LIN {X 0,Y 303.786,Z 846.921,A -85,B 0,C 180,E1 -15924.689,E2 -15924.689} C_VEL
LIN {X 0,Y 303.796,Z 848.766,A -85,B 0,C 180,E1 -15926.019,E2 -15926.019} C_VEL
LIN {X 0,Y 303.768,Z 850.119,A -85,B 0,C 180,E1 -15927.346,E2 -15927.346} C_VEL
LIN {X 0,Y 303.87,Z 851.06,A -85,B 0,C 180,E1 -15928.673,E2 -15928.673} C_VEL
LIN {X 0,Y 303.954,Z 851.584,A -85,B 0,C 180,E1 -15929.999,E2 -15929.999} C_VEL
LIN {X 0,Y 303.824,Z 851.641,A -85,B 0,C 180,E1 -15931.324,E2 -15931.324} C_VEL
LIN {X 0,Y 303.734,Z 851.272,A -85,B 0,C 180,E1 -15932.651,E2 -15932.651} C_VEL
LIN {X 0,Y 303.715,Z 850.5,A -85,B 0,C 180,E1 -15933.979,E2 -15933.979} C_VEL
LIN {X 0,Y 303.689,Z 848.909,A -85,B 0,C 180,E1 -15935.665,E2 -15935.665} C_VEL
LIN {X 0,Y 303.939,Z 845.59,A -85,B 0,C 180,E1 -15937.973,E2 -15937.973} C_VEL
LIN {X 0,Y 304.361,Z 841.592,A -85,B 0,C 180,E1 -15939.971,E2 -15939.971} C_VEL
LIN {X 0,Y 305.048,Z 836.47,A -85,B 0,C 180,E1 -15941.966,E2 -15941.966} C_VEL
LIN {X 0,Y 306.228,Z 830.072,A -85,B 0,C 180,E1 -15943.943,E2 -15943.943} C_VEL
LIN {X 0,Y 307.615,Z 822.158,A -85,B 0,C 180,E1 -15945.91,E2 -15945.91} C_VEL
LIN {X 0,Y 309.269,Z 812.287,A -85,B 0,C 180,E1 -15947.864,E2 -15947.864} C_VEL
LIN {X 0,Y 311.114,Z 802.166,A -85,B 0,C 180,E1 -15949.461,E2 -15949.461} C_VEL
LIN {X 0,Y 312.828,Z 792.253,A -85,B 0,C 180,E1 -15950.721,E2 -15950.721} C_VEL
LIN {X 0,Y 314.602,Z 779.923,A -85,B 0,C 180,E1 -15951.972,E2 -15951.972} C_VEL
LIN {X 0,Y 316.384,Z 766.923,A -85,B 0,C 180,E1 -15952.961,E2 -15952.961} C_VEL
LIN {X 0,Y 317.699,Z 753.709,A -85,B 0,C 180,E1 -15953.679,E2 -15953.679} C_VEL
LIN {X 0,Y 318.529,Z 740.017,A -85,B 0,C 180,E1 -15954.176,E2 -15954.176} C_VEL
LIN {X 0,Y 320.65,Z 684.229,A -85,B 0,C 180,E1 -15955.689,E2 -15955.689} C_VEL
LIN {X 0,Y 318.484,Z 666.248,A -85,B 0,C 180,E1 -15956.514,E2 -15956.514} C_VEL
LIN {X 0,Y 315.684,Z 649.939,A -85,B 0,C 180,E1 -15957.399,E2 -15957.399} C_VEL
LIN {X 0,Y 312.951,Z 638.201,A -85,B 0,C 180,E1 -15958.147,E2 -15958.147} C_VEL
LIN {X 0,Y 312.146,Z 635.73,A -85,B 0,C 180,E1 -15958.373,E2 -15958.373} C_VEL
LIN {X 0,Y 310.349,Z 626.488,A -85,B 0,C 180,E1 -15961.387,E2 -15961.387} C_VEL
LIN {X 0,Y 308.701,Z 619.358,A -85,B 0,C 180,E1 -15963.9,E2 -15963.9} C_VEL
LIN {X 0,Y 306.797,Z 612.092,A -85,B 0,C 180,E1 -15966.7,E2 -15966.7} C_VEL
LIN {X 0,Y 305.491,Z 607.435,A -85,B 0,C 180,E1 -15968.684,E2 -15968.684} C_VEL
LIN {X 0,Y 305.495,Z 607.433,A -85,B 0,C 180,E1 -15972.594,E2 -15972.594} C_VEL
LIN {X 0,Y 305.497,Z 607.431,A -85,B 0,C 180,E1 -15976.357,E2 -15976.357} C_VEL
LIN {X 0,Y 305.494,Z 607.433,A -85,B 0,C 180,E1 -15979.898,E2 -15979.898} C_VEL
LIN {X 0,Y 305.497,Z 607.426,A -85,B 0,C 180,E1 -15983.625,E2 -15983.625} C_VEL
LIN {X 0,Y 305.46,Z 607.431,A -85,B 0,C 180,E1 -15986.482,E2 -15986.482} C_VEL
LIN {X 0,Y 305.46,Z 607.432,A -85,B 0,C 180,E1 -15989.59,E2 -15989.59} C_VEL
LIN {X 0,Y 305.515,Z 607.427,A -85,B 0,C 180,E1 -15992.608,E2 -15992.608} C_VEL
LIN {X 0,Y 305.501,Z 607.428,A -85,B 0,C 180,E1 -15995.538,E2 -15995.538} C_VEL
LIN {X 0,Y 305.512,Z 607.423,A -85,B 0,C 180,E1 -15999.814,E2 -15999.814} C_VEL
LIN {X 0,Y 305.566,Z 607.418,A -85,B 0,C 180,E1 -16002.602,E2 -16002.602} C_VEL
LIN {X 0,Y 305.641,Z 607.408,A -85,B 0,C 180,E1 -16005.348,E2 -16005.348} C_VEL
LIN {X 0,Y 305.632,Z 607.414,A -85,B 0,C 180,E1 -16009.399,E2 -16009.399} C_VEL
LIN {X 0,Y 305.805,Z 607.392,A -85,B 0,C 180,E1 -16012.074,E2 -16012.074} C_VEL
LIN {X 0,Y 305.682,Z 607.406,A -85,B 0,C 180,E1 -16014.723,E2 -16014.723} C_VEL
LIN {X 0,Y 305.951,Z 607.373,A -85,B 0,C 180,E1 -16018.684,E2 -16018.684} C_VEL
LIN {X 0,Y 305.953,Z 607.376,A -85,B 0,C 180,E1 -16021.316,E2 -16021.316} C_VEL
LIN {X 0,Y 305.658,Z 607.553,A -85,B 0,C 180,E1 -16024.533,E2 -16024.533} C_VEL
LIN {X 0,Y 306.632,Z 610.635,A -85,B 0,C 180,E1 -16025.982,E2 -16025.982} C_VEL
LIN {X 0,Y 313.096,Z 622.289,A -85,B 0,C 180,E1 -16027.316,E2 -16027.316} C_VEL
LIN {X 0,Y 320.199,Z 637.232,A -85,B 0,C 180,E1 -16028.725,E2 -16028.725} C_VEL
LIN {X 0,Y 322.11,Z 641.956,A -85,B 0,C 180,E1 -16029.111,E2 -16029.111} C_VEL
LIN {X 0,Y 319.07,Z 715.822,A -85,B 0,C 180,E1 -16031.152,E2 -16031.152} C_VEL
LIN {X 0,Y 318.2,Z 728.923,A -85,B 0,C 180,E1 -16031.757,E2 -16031.757} C_VEL
LIN {X 0,Y 317.117,Z 741.244,A -85,B 0,C 180,E1 -16032.577,E2 -16032.577} C_VEL
LIN {X 0,Y 315.862,Z 751.913,A -85,B 0,C 180,E1 -16033.511,E2 -16033.511} C_VEL
LIN {X 0,Y 314.2,Z 763.939,A -85,B 0,C 180,E1 -16034.87,E2 -16034.87} C_VEL
LIN {X 0,Y 312.488,Z 774.225,A -85,B 0,C 180,E1 -16036.328,E2 -16036.328} C_VEL
LIN {X 0,Y 310.781,Z 783.569,A -85,B 0,C 180,E1 -16037.98,E2 -16037.98} C_VEL
LIN {X 0,Y 309.046,Z 792.453,A -85,B 0,C 180,E1 -16039.945,E2 -16039.945} C_VEL
LIN {X 0,Y 307.616,Z 799.149,A -85,B 0,C 180,E1 -16041.793,E2 -16041.793} C_VEL
LIN {X 0,Y 306.432,Z 805.122,A -85,B 0,C 180,E1 -16043.896,E2 -16043.896} C_VEL
LIN {X 0,Y 305.394,Z 810.016,A -85,B 0,C 180,E1 -16046.172,E2 -16046.172} C_VEL
LIN {X 0,Y 304.957,Z 812.136,A -85,B 0,C 180,E1 -16047.446,E2 -16047.446} C_VEL
LIN {X 0,Y 304.502,Z 814.135,A -85,B 0,C 180,E1 -16048.992,E2 -16048.992} C_VEL
LIN {X 0,Y 304,Z 815.985,A -85,B 0,C 180,E1 -16051.201,E2 -16051.201} C_VEL
LIN {X 0,Y 303.73,Z 816.702,A -85,B 0,C 180,E1 -16053.734,E2 -16053.734} C_VEL
LIN {X 0,Y 303.63,Z 816.128,A -85,B 0,C 180,E1 -16055.894,E2 -16055.894} C_VEL
LIN {X 0,Y 303.743,Z 814.383,A -85,B 0,C 180,E1 -16058.125,E2 -16058.125} C_VEL
LIN {X 0,Y 304.075,Z 811.449,A -85,B 0,C 180,E1 -16060.327,E2 -16060.327} C_VEL
LIN {X 0,Y 304.45,Z 807.575,A -85,B 0,C 180,E1 -16062.382,E2 -16062.382} C_VEL
LIN {X 0,Y 305.045,Z 802.499,A -85,B 0,C 180,E1 -16064.423,E2 -16064.423} C_VEL
LIN {X 0,Y 305.768,Z 796.24,A -85,B 0,C 180,E1 -16066.408,E2 -16066.408} C_VEL
LIN {X 0,Y 306.705,Z 788.58,A -85,B 0,C 180,E1 -16068.357,E2 -16068.357} C_VEL
LIN {X 0,Y 307.67,Z 780.998,A -85,B 0,C 180,E1 -16069.927,E2 -16069.927} C_VEL
LIN {X 0,Y 308.786,Z 771.91,A -85,B 0,C 180,E1 -16071.479,E2 -16071.479} C_VEL
LIN {X 0,Y 310.089,Z 760.631,A -85,B 0,C 180,E1 -16073.027,E2 -16073.027} C_VEL
LIN {X 0,Y 311.104,Z 749.624,A -85,B 0,C 180,E1 -16074.238,E2 -16074.238} C_VEL
LIN {X 0,Y 312.157,Z 737.533,A -85,B 0,C 180,E1 -16075.263,E2 -16075.263} C_VEL
LIN {X 0,Y 312.912,Z 724.139,A -85,B 0,C 180,E1 -16076.108,E2 -16076.108} C_VEL
LIN {X 0,Y 313.468,Z 711.355,A -85,B 0,C 180,E1 -16076.648,E2 -16076.648} C_VEL
LIN {X 0,Y 315.639,Z 635.414,A -85,B 0,C 180,E1 -16078.638,E2 -16078.638} C_VEL
LIN {X 0,Y 308.701,Z 615.889,A -85,B 0,C 180,E1 -16079.648,E2 -16079.648} C_VEL
LIN {X 0,Y 305.52,Z 607.516,A -85,B 0,C 180,E1 -16080.111,E2 -16080.111} C_VEL
LIN {X 0,Y 305.568,Z 607.425,A -85,B 0,C 180,E1 -16084.089,E2 -16084.089} C_VEL
LIN {X 0,Y 305.527,Z 607.428,A -85,B 0,C 180,E1 -16088.407,E2 -16088.407} C_VEL
LIN {X 0,Y 305.59,Z 607.416,A -85,B 0,C 180,E1 -16091.219,E2 -16091.219} C_VEL
LIN {X 0,Y 305.648,Z 607.409,A -85,B 0,C 180,E1 -16095.351,E2 -16095.351} C_VEL
LIN {X 0,Y 305.64,Z 607.41,A -85,B 0,C 180,E1 -16099.401,E2 -16099.401} C_VEL
LIN {X 0,Y 305.813,Z 607.391,A -85,B 0,C 180,E1 -16102.076,E2 -16102.076} C_VEL
LIN {X 0,Y 305.69,Z 607.407,A -85,B 0,C 180,E1 -16104.725,E2 -16104.725} C_VEL
LIN {X 0,Y 305.957,Z 607.375,A -85,B 0,C 180,E1 -16108.685,E2 -16108.685} C_VEL
LIN {X 0,Y 305.961,Z 607.37,A -85,B 0,C 180,E1 -16111.318,E2 -16111.318} C_VEL
LIN {X 0,Y 305.692,Z 607.404,A -85,B 0,C 180,E1 -16115.278,E2 -16115.278} C_VEL
LIN {X 0,Y 305.815,Z 607.388,A -85,B 0,C 180,E1 -16117.927,E2 -16117.927} C_VEL
LIN {X 0,Y 305.606,Z 607.414,A -85,B 0,C 180,E1 -16121.946,E2 -16121.946} C_VEL
LIN {X 0,Y 305.64,Z 607.413,A -85,B 0,C 180,E1 -16125.036,E2 -16125.036} C_VEL
LIN {X 0,Y 305.579,Z 607.416,A -85,B 0,C 180,E1 -16129.446,E2 -16129.446} C_VEL
LIN {X 0,Y 305.494,Z 607.433,A -85,B 0,C 180,E1 -16133.043,E2 -16133.043} C_VEL
LIN {X 0,Y 305.529,Z 607.424,A -85,B 0,C 180,E1 -16136.22,E2 -16136.22} C_VEL
LIN {X 0,Y 305.492,Z 607.434,A -85,B 0,C 180,E1 -16139.049,E2 -16139.049} C_VEL
LIN {X 0,Y 305.445,Z 607.432,A -85,B 0,C 180,E1 -16141.953,E2 -16141.953} C_VEL
LIN {X 0,Y 305.466,Z 607.433,A -85,B 0,C 180,E1 -16145.114,E2 -16145.114} C_VEL
LIN {X 0,Y 305.444,Z 607.434,A -85,B 0,C 180,E1 -16148.528,E2 -16148.528} C_VEL
LIN {X 0,Y 305.463,Z 607.432,A -85,B 0,C 180,E1 -16152.587,E2 -16152.587} C_VEL
LIN {X 0,Y 305.447,Z 607.433,A -85,B 0,C 180,E1 -16156.349,E2 -16156.349} C_VEL
LIN {X 0,Y 305.462,Z 607.431,A -85,B 0,C 180,E1 -16159.893,E2 -16159.893} C_VEL
LIN {X 0,Y 305.454,Z 607.429,A -85,B 0,C 180,E1 -16162.054,E2 -16162.054} C_VEL
LIN {X 0,Y 304.762,Z 607.519,A -85,B 0,C 180,E1 -16163.155,E2 -16163.155} C_VEL
LIN {X 0,Y 301.888,Z 607.875,A -85,B 0,C 180,E1 -16164.947,E2 -16164.947} C_VEL
LIN {X 0,Y 299.48,Z 608.175,A -85,B 0,C 180,E1 -16166.4,E2 -16166.4} C_VEL
LIN {X 0,Y 298.47,Z 608.306,A -85,B 0,C 180,E1 -16167.526,E2 -16167.526} C_VEL
LIN {X 0,Y 298.399,Z 608.313,A -85,B 0,C 180,E1 -16167.907,E2 -16167.907} C_VEL
LIN {X 0,Y 298.469,Z 608.307,A -85,B 0,C 180,E1 -16171.905,E2 -16171.905} C_VEL
LIN {X 0,Y 298.489,Z 608.301,A -85,B 0,C 180,E1 -16174.925,E2 -16174.925} C_VEL
LIN {X 0,Y 298.443,Z 608.306,A -85,B 0,C 180,E1 -16179.315,E2 -16179.315} C_VEL
LIN {X 0,Y 298.54,Z 608.292,A -85,B 0,C 180,E1 -16182.18,E2 -16182.18} C_VEL
LIN {X 0,Y 298.599,Z 608.282,A -85,B 0,C 180,E1 -16184.995,E2 -16184.995} C_VEL
LIN {X 0,Y 298.598,Z 608.286,A -85,B 0,C 180,E1 -16189.147,E2 -16189.147} C_VEL
LIN {X 0,Y 298.747,Z 608.272,A -85,B 0,C 180,E1 -16191.886,E2 -16191.886} C_VEL
LIN {X 0,Y 298.662,Z 608.28,A -85,B 0,C 180,E1 -16194.599,E2 -16194.599} C_VEL
LIN {X 0,Y 298.928,Z 608.245,A -85,B 0,C 180,E1 -16198.653,E2 -16198.653} C_VEL
LIN {X 0,Y 298.928,Z 608.242,A -85,B 0,C 180,E1 -16201.347,E2 -16201.347} C_VEL
LIN {X 0,Y 298.794,Z 608.264,A -85,B 0,C 180,E1 -16206.754,E2 -16206.754} C_VEL
LIN {X 0,Y 298.642,Z 608.282,A -85,B 0,C 180,E1 -16209.482,E2 -16209.482} C_VEL
LIN {X 0,Y 298.552,Z 608.292,A -85,B 0,C 180,E1 -16213.616,E2 -16213.616} C_VEL
LIN {X 0,Y 298.49,Z 608.303,A -85,B 0,C 180,E1 -16216.412,E2 -16216.412} C_VEL
LIN {X 0,Y 298.466,Z 608.304,A -85,B 0,C 180,E1 -16219.627,E2 -16219.627} C_VEL
LIN {X 0,Y 298.435,Z 608.307,A -85,B 0,C 180,E1 -16223.6,E2 -16223.6} C_VEL
LIN {X 0,Y 298.498,Z 608.303,A -85,B 0,C 180,E1 -16226.574,E2 -16226.574} C_VEL
LIN {X 0,Y 298.427,Z 608.309,A -85,B 0,C 180,E1 -16229.641,E2 -16229.641} C_VEL
LIN {X 0,Y 298.401,Z 608.316,A -85,B 0,C 180,E1 -16232.8,E2 -16232.8} C_VEL
LIN {X 0,Y 298.45,Z 608.311,A -85,B 0,C 180,E1 -16236.806,E2 -16236.806} C_VEL
LIN {X 0,Y 298.394,Z 608.317,A -85,B 0,C 180,E1 -16241.087,E2 -16241.087} C_VEL
LIN {X 0,Y 298.394,Z 608.318,A -85,B 0,C 180,E1 -16245.041,E2 -16245.041} C_VEL
LIN {X 0,Y 298.393,Z 608.317,A -85,B 0,C 180,E1 -16248.911,E2 -16248.911} C_VEL
LIN {X 0,Y 298.45,Z 608.311,A -85,B 0,C 180,E1 -16253.192,E2 -16253.192} C_VEL
LIN {X 0,Y 298.448,Z 608.42,A -85,B 0,C 180,E1 -16255.751,E2 -16255.751} C_VEL
LIN {X 0,Y 301.082,Z 620.831,A -85,B 0,C 180,E1 -16259.479,E2 -16259.479} C_VEL
LIN {X 0,Y 303.19,Z 630.91,A -85,B 0,C 180,E1 -16262.379,E2 -16262.379} C_VEL
LIN {X 0,Y 303.241,Z 633.696,A -85,B 0,C 180,E1 -16263.131,E2 -16263.131} C_VEL
LIN {X 0,Y 302.442,Z 639.311,A -85,B 0,C 180,E1 -16264.586,E2 -16264.586} C_VEL
LIN {X 0,Y 308.114,Z 684.772,A -85,B 0,C 180,E1 -16266.296,E2 -16266.296} C_VEL
LIN {X 0,Y 306.225,Z 749.237,A -85,B 0,C 180,E1 -16268.057,E2 -16268.057} C_VEL
LIN {X 0,Y 305.404,Z 762.213,A -85,B 0,C 180,E1 -16268.66,E2 -16268.66} C_VEL
LIN {X 0,Y 304.335,Z 774.343,A -85,B 0,C 180,E1 -16269.467,E2 -16269.467} C_VEL
LIN {X 0,Y 303.101,Z 786.172,A -85,B 0,C 180,E1 -16270.529,E2 -16270.529} C_VEL
LIN {X 0,Y 301.763,Z 797.631,A -85,B 0,C 180,E1 -16271.849,E2 -16271.849} C_VEL
LIN {X 0,Y 300.511,Z 808.02,A -85,B 0,C 180,E1 -16273.351,E2 -16273.351} C_VEL
LIN {X 0,Y 299.442,Z 817.358,A -85,B 0,C 180,E1 -16275.037,E2 -16275.037} C_VEL
LIN {X 0,Y 298.326,Z 826.437,A -85,B 0,C 180,E1 -16277.066,E2 -16277.066} C_VEL
LIN {X 0,Y 297.485,Z 833.693,A -85,B 0,C 180,E1 -16279.104,E2 -16279.104} C_VEL
LIN {X 0,Y 297.018,Z 839.454,A -85,B 0,C 180,E1 -16281.151,E2 -16281.151} C_VEL
LIN {X 0,Y 296.789,Z 843.951,A -85,B 0,C 180,E1 -16283.199,E2 -16283.199} C_VEL
LIN {X 0,Y 296.701,Z 846.302,A -85,B 0,C 180,E1 -16284.562,E2 -16284.562} C_VEL
LIN {X 0,Y 296.727,Z 848.202,A -85,B 0,C 180,E1 -16285.924,E2 -16285.924} C_VEL
LIN {X 0,Y 296.688,Z 849.596,A -85,B 0,C 180,E1 -16287.283,E2 -16287.283} C_VEL
LIN {X 0,Y 296.778,Z 850.566,A -85,B 0,C 180,E1 -16288.642,E2 -16288.642} C_VEL
LIN {X 0,Y 296.867,Z 851.119,A -85,B 0,C 180,E1 -16289.999,E2 -16289.999} C_VEL
LIN {X 0,Y 296.73,Z 851.23,A -85,B 0,C 180,E1 -16291.356,E2 -16291.356} C_VEL
LIN {X 0,Y 296.653,Z 850.888,A -85,B 0,C 180,E1 -16292.714,E2 -16292.714} C_VEL
LIN {X 0,Y 296.626,Z 850.14,A -85,B 0,C 180,E1 -16294.074,E2 -16294.074} C_VEL
LIN {X 0,Y 296.606,Z 848.802,A -85,B 0,C 180,E1 -16295.625,E2 -16295.625} C_VEL
LIN {X 0,Y 296.873,Z 845.348,A -85,B 0,C 180,E1 -16298.164,E2 -16298.164} C_VEL
LIN {X 0,Y 297.348,Z 841.428,A -85,B 0,C 180,E1 -16300.209,E2 -16300.209} C_VEL
LIN {X 0,Y 298.067,Z 836.374,A -85,B 0,C 180,E1 -16302.25,E2 -16302.25} C_VEL
LIN {X 0,Y 299.332,Z 830.045,A -85,B 0,C 180,E1 -16304.271,E2 -16304.271} C_VEL
LIN {X 0,Y 300.792,Z 822.225,A -85,B 0,C 180,E1 -16306.281,E2 -16306.281} C_VEL
LIN {X 0,Y 302.536,Z 812.502,A -85,B 0,C 180,E1 -16308.275,E2 -16308.275} C_VEL
LIN {X 0,Y 304.45,Z 802.56,A -85,B 0,C 180,E1 -16309.905,E2 -16309.905} C_VEL
LIN {X 0,Y 306.493,Z 791.545,A -85,B 0,C 180,E1 -16311.346,E2 -16311.346} C_VEL
LIN {X 0,Y 308.093,Z 780.913,A -85,B 0,C 180,E1 -16312.461,E2 -16312.461} C_VEL
LIN {X 0,Y 310.062,Z 767.228,A -85,B 0,C 180,E1 -16313.545,E2 -16313.545} C_VEL
LIN {X 0,Y 311.36,Z 755.244,A -85,B 0,C 180,E1 -16314.236,E2 -16314.236} C_VEL
LIN {X 0,Y 312.309,Z 741.359,A -85,B 0,C 180,E1 -16314.778,E2 -16314.778} C_VEL
LIN {X 0,Y 314.649,Z 685.473,A -85,B 0,C 180,E1 -16316.333,E2 -16316.333} C_VEL
LIN {X 0,Y 312.673,Z 668.247,A -85,B 0,C 180,E1 -16317.155,E2 -16317.155} C_VEL
LIN {X 0,Y 309.901,Z 651.84,A -85,B 0,C 180,E1 -16318.07,E2 -16318.07} C_VEL
LIN {X 0,Y 307.431,Z 641.003,A -85,B 0,C 180,E1 -16318.792,E2 -16318.792} C_VEL
LIN {X 0,Y 304.991,Z 635.218,A -85,B 0,C 180,E1 -16319.361,E2 -16319.361} C_VEL
LIN {X 0,Y 303.047,Z 625.874,A -85,B 0,C 180,E1 -16322.577,E2 -16322.577} C_VEL
LIN {X 0,Y 301.051,Z 617.638,A -85,B 0,C 180,E1 -16325.704,E2 -16325.704} C_VEL
LIN {X 0,Y 298.78,Z 609.723,A -85,B 0,C 180,E1 -16329.082,E2 -16329.082} C_VEL
LIN {X 0,Y 298.43,Z 608.316,A -85,B 0,C 180,E1 -16329.809,E2 -16329.809} C_VEL
LIN {X 0,Y 298.454,Z 608.311,A -85,B 0,C 180,E1 -16333.114,E2 -16333.114} C_VEL
LIN {X 0,Y 298.462,Z 608.307,A -85,B 0,C 180,E1 -16336.931,E2 -16336.931} C_VEL
LIN {X 0,Y 298.434,Z 608.307,A -85,B 0,C 180,E1 -16340.996,E2 -16340.996} C_VEL
LIN {X 0,Y 298.428,Z 608.307,A -85,B 0,C 180,E1 -16343.931,E2 -16343.931} C_VEL
LIN {X 0,Y 298.393,Z 608.312,A -85,B 0,C 180,E1 -16347.981,E2 -16347.981} C_VEL
LIN {X 0,Y 298.457,Z 608.301,A -85,B 0,C 180,E1 -16351.903,E2 -16351.903} C_VEL
LIN {X 0,Y 298.478,Z 608.302,A -85,B 0,C 180,E1 -16354.923,E2 -16354.923} C_VEL
LIN {X 0,Y 298.451,Z 608.303,A -85,B 0,C 180,E1 -16359.315,E2 -16359.315} C_VEL
LIN {X 0,Y 298.53,Z 608.295,A -85,B 0,C 180,E1 -16362.179,E2 -16362.179} C_VEL
LIN {X 0,Y 298.585,Z 608.287,A -85,B 0,C 180,E1 -16364.994,E2 -16364.994} C_VEL
LIN {X 0,Y 298.587,Z 608.292,A -85,B 0,C 180,E1 -16369.146,E2 -16369.146} C_VEL
LIN {X 0,Y 298.75,Z 608.272,A -85,B 0,C 180,E1 -16371.886,E2 -16371.886} C_VEL
LIN {X 0,Y 298.653,Z 608.281,A -85,B 0,C 180,E1 -16374.599,E2 -16374.599} C_VEL
LIN {X 0,Y 298.917,Z 608.249,A -85,B 0,C 180,E1 -16378.653,E2 -16378.653} C_VEL
LIN {X 0,Y 298.92,Z 608.252,A -85,B 0,C 180,E1 -16381.347,E2 -16381.347} C_VEL
LIN {X 0,Y 298.71,Z 608.484,A -85,B 0,C 180,E1 -16383.541,E2 -16383.541} C_VEL
LIN {X 0,Y 299.47,Z 611.352,A -85,B 0,C 180,E1 -16384.901,E2 -16384.901} C_VEL
LIN {X 0,Y 301.738,Z 615.054,A -85,B 0,C 180,E1 -16385.408,E2 -16385.408} C_VEL
LIN {X 0,Y 307.159,Z 624.505,A -85,B 0,C 180,E1 -16386.569,E2 -16386.569} C_VEL
LIN {X 0,Y 314.123,Z 639.09,A -85,B 0,C 180,E1 -16388.029,E2 -16388.029} C_VEL
LIN {X 0,Y 316.129,Z 643.93,A -85,B 0,C 180,E1 -16388.446,E2 -16388.446} C_VEL
LIN {X 0,Y 312.959,Z 716.358,A -85,B 0,C 180,E1 -16390.513,E2 -16390.513} C_VEL
LIN {X 0,Y 312.01,Z 729.333,A -85,B 0,C 180,E1 -16391.12,E2 -16391.12} C_VEL
LIN {X 0,Y 310.85,Z 742.08,A -85,B 0,C 180,E1 -16391.989,E2 -16391.989} C_VEL
LIN {X 0,Y 309.566,Z 752.553,A -85,B 0,C 180,E1 -16392.929,E2 -16392.929} C_VEL
LIN {X 0,Y 307.93,Z 763.714,A -85,B 0,C 180,E1 -16394.202,E2 -16394.202} C_VEL
LIN {X 0,Y 306.153,Z 774.096,A -85,B 0,C 180,E1 -16395.684,E2 -16395.684} C_VEL
LIN {X 0,Y 304.529,Z 782.271,A -85,B 0,C 180,E1 -16397.112,E2 -16397.112} C_VEL
LIN {X 0,Y 302.774,Z 790.87,A -85,B 0,C 180,E1 -16398.964,E2 -16398.964} C_VEL
LIN {X 0,Y 301.102,Z 798.39,A -85,B 0,C 180,E1 -16400.996,E2 -16400.996} C_VEL
LIN {X 0,Y 299.99,Z 803.587,A -85,B 0,C 180,E1 -16402.74,E2 -16402.74} C_VEL
LIN {X 0,Y 298.844,Z 808.961,A -85,B 0,C 180,E1 -16405.044,E2 -16405.044} C_VEL
LIN {X 0,Y 297.906,Z 812.957,A -85,B 0,C 180,E1 -16407.389,E2 -16407.389} C_VEL
LIN {X 0,Y 297.229,Z 815.585,A -85,B 0,C 180,E1 -16409.772,E2 -16409.772} C_VEL
LIN {X 0,Y 296.859,Z 816.722,A -85,B 0,C 180,E1 -16411.542,E2 -16411.542} C_VEL
LIN {X 0,Y 296.619,Z 817.11,A -85,B 0,C 180,E1 -16413.978,E2 -16413.978} C_VEL
LIN {X 0,Y 296.547,Z 816.232,A -85,B 0,C 180,E1 -16416.333,E2 -16416.333} C_VEL
LIN {X 0,Y 296.72,Z 814.22,A -85,B 0,C 180,E1 -16418.593,E2 -16418.593} C_VEL
LIN {X 0,Y 297.06,Z 811.101,A -85,B 0,C 180,E1 -16420.796,E2 -16420.796} C_VEL
LIN {X 0,Y 297.501,Z 806.92,A -85,B 0,C 180,E1 -16422.921,E2 -16422.921} C_VEL
LIN {X 0,Y 298.129,Z 801.56,A -85,B 0,C 180,E1 -16425.008,E2 -16425.008} C_VEL
LIN {X 0,Y 298.929,Z 795.017,A -85,B 0,C 180,E1 -16427.017,E2 -16427.017} C_VEL
LIN {X 0,Y 299.954,Z 786.927,A -85,B 0,C 180,E1 -16429.003,E2 -16429.003} C_VEL
LIN {X 0,Y 301.06,Z 778.449,A -85,B 0,C 180,E1 -16430.695,E2 -16430.695} C_VEL
LIN {X 0,Y 302.333,Z 767.866,A -85,B 0,C 180,E1 -16432.406,E2 -16432.406} C_VEL
LIN {X 0,Y 303.664,Z 756.132,A -85,B 0,C 180,E1 -16433.9,E2 -16433.9} C_VEL
LIN {X 0,Y 304.809,Z 744.207,A -85,B 0,C 180,E1 -16435.092,E2 -16435.092} C_VEL
LIN {X 0,Y 305.749,Z 731.208,A -85,B 0,C 180,E1 -16436.069,E2 -16436.069} C_VEL
LIN {X 0,Y 306.436,Z 718.25,A -85,B 0,C 180,E1 -16436.767,E2 -16436.767} C_VEL
LIN {X 0,Y 306.93,Z 704.012,A -85,B 0,C 180,E1 -16437.237,E2 -16437.237} C_VEL
LIN {X 0,Y 308.934,Z 636.819,A -85,B 0,C 180,E1 -16439.025,E2 -16439.025} C_VEL
LIN {X 0,Y 301.755,Z 616.857,A -85,B 0,C 180,E1 -16440.097,E2 -16440.097} C_VEL
LIN {X 0,Y 298.513,Z 608.56,A -85,B 0,C 180,E1 -16440.577,E2 -16440.577} C_VEL
LIN {X 0,Y 298.458,Z 608.306,A -85,B 0,C 180,E1 -16440.606,E2 -16440.606} C_VEL
LIN {X 0,Y 298.475,Z 608.304,A -85,B 0,C 180,E1 -16443.478,E2 -16443.478} C_VEL
LIN {X 0,Y 298.433,Z 608.309,A -85,B 0,C 180,E1 -16446.699,E2 -16446.699} C_VEL
LIN {X 0,Y 298.541,Z 608.295,A -85,B 0,C 180,E1 -16450.759,E2 -16450.759} C_VEL
LIN {X 0,Y 298.592,Z 608.288,A -85,B 0,C 180,E1 -16454.996,E2 -16454.996} C_VEL
LIN {X 0,Y 298.595,Z 608.288,A -85,B 0,C 180,E1 -16459.148,E2 -16459.148} C_VEL
LIN {X 0,Y 298.758,Z 608.269,A -85,B 0,C 180,E1 -16461.887,E2 -16461.887} C_VEL
LIN {X 0,Y 298.661,Z 608.284,A -85,B 0,C 180,E1 -16464.6,E2 -16464.6} C_VEL
LIN {X 0,Y 298.923,Z 608.251,A -85,B 0,C 180,E1 -16468.654,E2 -16468.654} C_VEL
LIN {X 0,Y 298.927,Z 608.246,A -85,B 0,C 180,E1 -16471.349,E2 -16471.349} C_VEL
LIN {X 0,Y 298.663,Z 608.279,A -85,B 0,C 180,E1 -16475.402,E2 -16475.402} C_VEL
LIN {X 0,Y 298.76,Z 608.268,A -85,B 0,C 180,E1 -16478.115,E2 -16478.115} C_VEL
LIN {X 0,Y 298.556,Z 608.293,A -85,B 0,C 180,E1 -16482.233,E2 -16482.233} C_VEL
LIN {X 0,Y 298.608,Z 608.288,A -85,B 0,C 180,E1 -16485.21,E2 -16485.21} C_VEL
LIN {X 0,Y 298.542,Z 608.294,A -85,B 0,C 180,E1 -16489.244,E2 -16489.244} C_VEL
LIN {X 0,Y 298.461,Z 608.305,A -85,B 0,C 180,E1 -16493.599,E2 -16493.599} C_VEL
LIN {X 0,Y 298.488,Z 608.302,A -85,B 0,C 180,E1 -16496.576,E2 -16496.576} C_VEL
LIN {X 0,Y 298.42,Z 608.309,A -85,B 0,C 180,E1 -16499.642,E2 -16499.642} C_VEL
LIN {X 0,Y 298.398,Z 608.312,A -85,B 0,C 180,E1 -16502.801,E2 -16502.801} C_VEL
LIN {X 0,Y 298.448,Z 608.305,A -85,B 0,C 180,E1 -16506.808,E2 -16506.808} C_VEL
LIN {X 0,Y 298.392,Z 608.316,A -85,B 0,C 180,E1 -16511.089,E2 -16511.089} C_VEL
LIN {X 0,Y 298.393,Z 608.315,A -85,B 0,C 180,E1 -16515.042,E2 -16515.042} C_VEL
LIN {X 0,Y 298.392,Z 608.312,A -85,B 0,C 180,E1 -16518.913,E2 -16518.913} C_VEL
LIN {X 0,Y 298.451,Z 608.302,A -85,B 0,C 180,E1 -16523.193,E2 -16523.193} C_VEL
LIN {X 0,Y 298.401,Z 608.311,A -85,B 0,C 180,E1 -16527.201,E2 -16527.201} C_VEL
LIN {X 0,Y 298.399,Z 608.313,A -85,B 0,C 180,E1 -16527.907,E2 -16527.907} C_VEL
LIN {X 0,Y 297.766,Z 608.395,A -85,B 0,C 180,E1 -16529.033,E2 -16529.033} C_VEL
LIN {X 0,Y 294.944,Z 608.746,A -85,B 0,C 180,E1 -16530.867,E2 -16530.867} C_VEL
LIN {X 0,Y 292.534,Z 609.043,A -85,B 0,C 180,E1 -16532.356,E2 -16532.356} C_VEL
LIN {X 0,Y 291.5,Z 609.175,A -85,B 0,C 180,E1 -16533.508,E2 -16533.508} C_VEL
LIN {X 0,Y 291.417,Z 609.181,A -85,B 0,C 180,E1 -16533.899,E2 -16533.899} C_VEL
LIN {X 0,Y 291.38,Z 609.187,A -85,B 0,C 180,E1 -16537.3,E2 -16537.3} C_VEL
LIN {X 0,Y 291.464,Z 609.173,A -85,B 0,C 180,E1 -16540.271,E2 -16540.271} C_VEL
LIN {X 0,Y 291.546,Z 609.16,A -85,B 0,C 180,E1 -16544.635,E2 -16544.635} C_VEL
LIN {X 0,Y 291.542,Z 609.165,A -85,B 0,C 180,E1 -16548.881,E2 -16548.881} C_VEL
LIN {X 0,Y 291.694,Z 609.149,A -85,B 0,C 180,E1 -16551.688,E2 -16551.688} C_VEL
LIN {X 0,Y 291.633,Z 609.157,A -85,B 0,C 180,E1 -16554.469,E2 -16554.469} C_VEL
LIN {X 0,Y 291.894,Z 609.121,A -85,B 0,C 180,E1 -16558.621,E2 -16558.621} C_VEL
LIN {X 0,Y 291.895,Z 609.117,A -85,B 0,C 180,E1 -16561.38,E2 -16561.38} C_VEL
LIN {X 0,Y 291.742,Z 609.142,A -85,B 0,C 180,E1 -16566.918,E2 -16566.918} C_VEL
LIN {X 0,Y 291.582,Z 609.162,A -85,B 0,C 180,E1 -16569.714,E2 -16569.714} C_VEL
LIN {X 0,Y 291.522,Z 609.169,A -85,B 0,C 180,E1 -16573.951,E2 -16573.951} C_VEL
LIN {X 0,Y 291.435,Z 609.181,A -85,B 0,C 180,E1 -16576.821,E2 -16576.821} C_VEL
LIN {X 0,Y 291.43,Z 609.181,A -85,B 0,C 180,E1 -16579.86,E2 -16579.86} C_VEL
LIN {X 0,Y 291.39,Z 609.187,A -85,B 0,C 180,E1 -16584.206,E2 -16584.206} C_VEL
LIN {X 0,Y 291.432,Z 609.181,A -85,B 0,C 180,E1 -16587.271,E2 -16587.271} C_VEL
LIN {X 0,Y 291.344,Z 609.194,A -85,B 0,C 180,E1 -16590.436,E2 -16590.436} C_VEL
LIN {X 0,Y 291.351,Z 609.19,A -85,B 0,C 180,E1 -16593.698,E2 -16593.698} C_VEL
LIN {X 0,Y 291.378,Z 609.189,A -85,B 0,C 180,E1 -16597.252,E2 -16597.252} C_VEL
LIN {X 0,Y 291.339,Z 609.195,A -85,B 0,C 180,E1 -16600.642,E2 -16600.642} C_VEL
LIN {X 0,Y 291.319,Z 609.196,A -85,B 0,C 180,E1 -16604.397,E2 -16604.397} C_VEL
LIN {X 0,Y 291.333,Z 609.193,A -85,B 0,C 180,E1 -16608.403,E2 -16608.403} C_VEL
LIN {X 0,Y 291.353,Z 609.195,A -85,B 0,C 180,E1 -16611.157,E2 -16611.157} C_VEL
LIN {X 0,Y 291.366,Z 609.191,A -85,B 0,C 180,E1 -16614.625,E2 -16614.625} C_VEL
LIN {X 0,Y 291.398,Z 609.262,A -85,B 0,C 180,E1 -16615.359,E2 -16615.359} C_VEL
LIN {X 0,Y 294.132,Z 622.193,A -85,B 0,C 180,E1 -16619.338,E2 -16619.338} C_VEL
LIN {X 0,Y 296.298,Z 632.778,A -85,B 0,C 180,E1 -16622.448,E2 -16622.448} C_VEL
LIN {X 0,Y 295.585,Z 638.984,A -85,B 0,C 180,E1 -16624.111,E2 -16624.111} C_VEL
LIN {X 0,Y 301.358,Z 684.637,A -85,B 0,C 180,E1 -16625.874,E2 -16625.874} C_VEL
LIN {X 0,Y 299.428,Z 748.677,A -85,B 0,C 180,E1 -16627.668,E2 -16627.668} C_VEL
LIN {X 0,Y 298.544,Z 762.417,A -85,B 0,C 180,E1 -16628.326,E2 -16628.326} C_VEL
LIN {X 0,Y 297.445,Z 774.363,A -85,B 0,C 180,E1 -16629.15,E2 -16629.15} C_VEL
LIN {X 0,Y 296.173,Z 786.089,A -85,B 0,C 180,E1 -16630.235,E2 -16630.235} C_VEL
LIN {X 0,Y 294.813,Z 797.495,A -85,B 0,C 180,E1 -16631.586,E2 -16631.586} C_VEL
LIN {X 0,Y 293.525,Z 807.823,A -85,B 0,C 180,E1 -16633.122,E2 -16633.122} C_VEL
LIN {X 0,Y 292.3,Z 817.959,A -85,B 0,C 180,E1 -16635.019,E2 -16635.019} C_VEL
LIN {X 0,Y 291.192,Z 826.858,A -85,B 0,C 180,E1 -16637.098,E2 -16637.098} C_VEL
LIN {X 0,Y 290.367,Z 833.92,A -85,B 0,C 180,E1 -16639.187,E2 -16639.187} C_VEL
LIN {X 0,Y 289.865,Z 840.384,A -85,B 0,C 180,E1 -16641.634,E2 -16641.634} C_VEL
LIN {X 0,Y 289.676,Z 845.201,A -85,B 0,C 180,E1 -16644.115,E2 -16644.115} C_VEL
LIN {X 0,Y 289.659,Z 847.622,A -85,B 0,C 180,E1 -16645.824,E2 -16645.824} C_VEL
LIN {X 0,Y 289.611,Z 849.074,A -85,B 0,C 180,E1 -16647.217,E2 -16647.217} C_VEL
LIN {X 0,Y 289.686,Z 850.071,A -85,B 0,C 180,E1 -16648.608,E2 -16648.608} C_VEL
LIN {X 0,Y 289.78,Z 850.652,A -85,B 0,C 180,E1 -16649.998,E2 -16649.998} C_VEL
LIN {X 0,Y 289.637,Z 850.805,A -85,B 0,C 180,E1 -16651.389,E2 -16651.389} C_VEL
LIN {X 0,Y 289.574,Z 850.507,A -85,B 0,C 180,E1 -16652.781,E2 -16652.781} C_VEL
LIN {X 0,Y 289.539,Z 849.79,A -85,B 0,C 180,E1 -16654.174,E2 -16654.174} C_VEL
LIN {X 0,Y 289.517,Z 848.668,A -85,B 0,C 180,E1 -16655.571,E2 -16655.571} C_VEL
LIN {X 0,Y 289.711,Z 846.172,A -85,B 0,C 180,E1 -16657.666,E2 -16657.666} C_VEL
LIN {X 0,Y 290.12,Z 842.665,A -85,B 0,C 180,E1 -16659.761,E2 -16659.761} C_VEL
LIN {X 0,Y 290.8,Z 838.067,A -85,B 0,C 180,E1 -16661.853,E2 -16661.853} C_VEL
LIN {X 0,Y 292.185,Z 831.195,A -85,B 0,C 180,E1 -16664.272,E2 -16664.272} C_VEL
LIN {X 0,Y 293.665,Z 823.739,A -85,B 0,C 180,E1 -16666.33,E2 -16666.33} C_VEL
LIN {X 0,Y 295.453,Z 814.554,A -85,B 0,C 180,E1 -16668.37,E2 -16668.37} C_VEL
LIN {X 0,Y 297.397,Z 805.168,A -85,B 0,C 180,E1 -16670.037,E2 -16670.037} C_VEL
LIN {X 0,Y 299.356,Z 794.812,A -85,B 0,C 180,E1 -16671.518,E2 -16671.518} C_VEL
LIN {X 0,Y 301.294,Z 783.46,A -85,B 0,C 180,E1 -16672.816,E2 -16672.816} C_VEL
LIN {X 0,Y 303.338,Z 770.81,A -85,B 0,C 180,E1 -16673.918,E2 -16673.918} C_VEL
LIN {X 0,Y 304.98,Z 757.431,A -85,B 0,C 180,E1 -16674.777,E2 -16674.777} C_VEL
LIN {X 0,Y 306.045,Z 744.363,A -85,B 0,C 180,E1 -16675.366,E2 -16675.366} C_VEL
LIN {X 0,Y 308.687,Z 686.564,A -85,B 0,C 180,E1 -16677.022,E2 -16677.022} C_VEL
LIN {X 0,Y 306.669,Z 668.174,A -85,B 0,C 180,E1 -16677.923,E2 -16677.923} C_VEL
LIN {X 0,Y 303.351,Z 649.432,A -85,B 0,C 180,E1 -16679.064,E2 -16679.064} C_VEL
LIN {X 0,Y 301.891,Z 643.671,A -85,B 0,C 180,E1 -16679.488,E2 -16679.488} C_VEL
LIN {X 0,Y 297.766,Z 634.536,A -85,B 0,C 180,E1 -16680.487,E2 -16680.487} C_VEL
LIN {X 0,Y 295.599,Z 624.645,A -85,B 0,C 180,E1 -16684.124,E2 -16684.124} C_VEL
LIN {X 0,Y 293.554,Z 616.786,A -85,B 0,C 180,E1 -16687.356,E2 -16687.356} C_VEL
LIN {X 0,Y 291.382,Z 609.192,A -85,B 0,C 180,E1 -16690.922,E2 -16690.922} C_VEL
LIN {X 0,Y 291.372,Z 609.192,A -85,B 0,C 180,E1 -16694.384,E2 -16694.384} C_VEL
LIN {X 0,Y 291.383,Z 609.188,A -85,B 0,C 180,E1 -16698.389,E2 -16698.389} C_VEL
LIN {X 0,Y 291.382,Z 609.186,A -85,B 0,C 180,E1 -16701.163,E2 -16701.163} C_VEL
LIN {X 0,Y 291.38,Z 609.191,A -85,B 0,C 180,E1 -16704.628,E2 -16704.628} C_VEL
LIN {X 0,Y 291.369,Z 609.186,A -85,B 0,C 180,E1 -16707.95,E2 -16707.95} C_VEL
LIN {X 0,Y 291.376,Z 609.181,A -85,B 0,C 180,E1 -16711.157,E2 -16711.157} C_VEL
LIN {X 0,Y 291.409,Z 609.178,A -85,B 0,C 180,E1 -16714.271,E2 -16714.271} C_VEL
LIN {X 0,Y 291.381,Z 609.184,A -85,B 0,C 180,E1 -16717.299,E2 -16717.299} C_VEL
LIN {X 0,Y 291.451,Z 609.177,A -85,B 0,C 180,E1 -16720.269,E2 -16720.269} C_VEL
LIN {X 0,Y 291.547,Z 609.165,A -85,B 0,C 180,E1 -16724.623,E2 -16724.623} C_VEL
LIN {X 0,Y 291.531,Z 609.172,A -85,B 0,C 180,E1 -16728.88,E2 -16728.88} C_VEL
LIN {X 0,Y 291.701,Z 609.151,A -85,B 0,C 180,E1 -16731.688,E2 -16731.688} C_VEL
LIN {X 0,Y 291.624,Z 609.157,A -85,B 0,C 180,E1 -16734.468,E2 -16734.468} C_VEL
LIN {X 0,Y 291.883,Z 609.126,A -85,B 0,C 180,E1 -16738.62,E2 -16738.62} C_VEL
LIN {X 0,Y 291.886,Z 609.129,A -85,B 0,C 180,E1 -16741.38,E2 -16741.38} C_VEL
LIN {X 0,Y 291.841,Z 609.326,A -85,B 0,C 180,E1 -16742.415,E2 -16742.415} C_VEL
LIN {X 0,Y 292.333,Z 612.029,A -85,B 0,C 180,E1 -16743.726,E2 -16743.726} C_VEL
LIN {X 0,Y 294.534,Z 615.665,A -85,B 0,C 180,E1 -16744.253,E2 -16744.253} C_VEL
LIN {X 0,Y 300.016,Z 624.602,A -85,B 0,C 180,E1 -16745.511,E2 -16745.511} C_VEL
LIN {X 0,Y 305.688,Z 635.647,A -85,B 0,C 180,E1 -16746.766,E2 -16746.766} C_VEL
LIN {X 0,Y 310.282,Z 646.104,A -85,B 0,C 180,E1 -16747.777,E2 -16747.777} C_VEL
LIN {X 0,Y 306.949,Z 716.449,A -85,B 0,C 180,E1 -16749.808,E2 -16749.808} C_VEL
LIN {X 0,Y 305.95,Z 729.781,A -85,B 0,C 180,E1 -16750.445,E2 -16750.445} C_VEL
LIN {X 0,Y 304.755,Z 742.154,A -85,B 0,C 180,E1 -16751.304,E2 -16751.304} C_VEL
LIN {X 0,Y 303.424,Z 752.355,A -85,B 0,C 180,E1 -16752.225,E2 -16752.225} C_VEL
LIN {X 0,Y 301.732,Z 763.23,A -85,B 0,C 180,E1 -16753.469,E2 -16753.469} C_VEL
LIN {X 0,Y 299.959,Z 773.466,A -85,B 0,C 180,E1 -16754.935,E2 -16754.935} C_VEL
LIN {X 0,Y 298.166,Z 782.055,A -85,B 0,C 180,E1 -16756.43,E2 -16756.43} C_VEL
LIN {X 0,Y 296.235,Z 791.097,A -85,B 0,C 180,E1 -16758.388,E2 -16758.388} C_VEL
LIN {X 0,Y 294.319,Z 799.176,A -85,B 0,C 180,E1 -16760.623,E2 -16760.623} C_VEL
LIN {X 0,Y 293.047,Z 804.699,A -85,B 0,C 180,E1 -16762.564,E2 -16762.564} C_VEL
LIN {X 0,Y 291.84,Z 809.915,A -85,B 0,C 180,E1 -16764.925,E2 -16764.925} C_VEL
LIN {X 0,Y 290.862,Z 813.726,A -85,B 0,C 180,E1 -16767.328,E2 -16767.328} C_VEL
LIN {X 0,Y 290.248,Z 815.905,A -85,B 0,C 180,E1 -16769.347,E2 -16769.347} C_VEL
LIN {X 0,Y 289.742,Z 817.348,A -85,B 0,C 180,E1 -16771.905,E2 -16771.905} C_VEL
LIN {X 0,Y 289.534,Z 817.439,A -85,B 0,C 180,E1 -16774.385,E2 -16774.385} C_VEL
LIN {X 0,Y 289.481,Z 816.312,A -85,B 0,C 180,E1 -16776.761,E2 -16776.761} C_VEL
LIN {X 0,Y 289.706,Z 813.998,A -85,B 0,C 180,E1 -16779.104,E2 -16779.104} C_VEL
LIN {X 0,Y 290.065,Z 810.649,A -85,B 0,C 180,E1 -16781.317,E2 -16781.317} C_VEL
LIN {X 0,Y 290.557,Z 806.187,A -85,B 0,C 180,E1 -16783.48,E2 -16783.48} C_VEL
LIN {X 0,Y 291.376,Z 799.617,A -85,B 0,C 180,E1 -16785.904,E2 -16785.904} C_VEL
LIN {X 0,Y 292.121,Z 793.654,A -85,B 0,C 180,E1 -16787.654,E2 -16787.654} C_VEL
LIN {X 0,Y 293.261,Z 785.186,A -85,B 0,C 180,E1 -16789.682,E2 -16789.682} C_VEL
LIN {X 0,Y 294.572,Z 775.223,A -85,B 0,C 180,E1 -16791.579,E2 -16791.579} C_VEL
LIN {X 0,Y 295.877,Z 764.446,A -85,B 0,C 180,E1 -16793.228,E2 -16793.228} C_VEL
LIN {X 0,Y 297.184,Z 752.378,A -85,B 0,C 180,E1 -16794.674,E2 -16794.674} C_VEL
LIN {X 0,Y 298.353,Z 740.206,A -85,B 0,C 180,E1 -16795.806,E2 -16795.806} C_VEL
LIN {X 0,Y 299.236,Z 727.177,A -85,B 0,C 180,E1 -16796.704,E2 -16796.704} C_VEL
LIN {X 0,Y 299.869,Z 713.937,A -85,B 0,C 180,E1 -16797.333,E2 -16797.333} C_VEL
LIN {X 0,Y 302.223,Z 638.409,A -85,B 0,C 180,E1 -16799.425,E2 -16799.425} C_VEL
LIN {X 0,Y 295.26,Z 619.044,A -85,B 0,C 180,E1 -16800.496,E2 -16800.496} C_VEL
LIN {X 0,Y 291.479,Z 609.704,A -85,B 0,C 180,E1 -16801.062,E2 -16801.062} C_VEL
LIN {X 0,Y 291.422,Z 609.182,A -85,B 0,C 180,E1 -16801.11,E2 -16801.11} C_VEL
LIN {X 0,Y 291.411,Z 609.186,A -85,B 0,C 180,E1 -16804.273,E2 -16804.273} C_VEL
LIN {X 0,Y 291.387,Z 609.186,A -85,B 0,C 180,E1 -16807.302,E2 -16807.302} C_VEL
LIN {X 0,Y 291.461,Z 609.181,A -85,B 0,C 180,E1 -16810.272,E2 -16810.272} C_VEL
LIN {X 0,Y 291.554,Z 609.167,A -85,B 0,C 180,E1 -16814.625,E2 -16814.625} C_VEL
LIN {X 0,Y 291.538,Z 609.168,A -85,B 0,C 180,E1 -16818.882,E2 -16818.882} C_VEL
LIN {X 0,Y 291.709,Z 609.146,A -85,B 0,C 180,E1 -16821.69,E2 -16821.69} C_VEL
LIN {X 0,Y 291.632,Z 609.16,A -85,B 0,C 180,E1 -16824.47,E2 -16824.47} C_VEL
LIN {X 0,Y 291.89,Z 609.128,A -85,B 0,C 180,E1 -16828.622,E2 -16828.622} C_VEL
LIN {X 0,Y 291.894,Z 609.123,A -85,B 0,C 180,E1 -16831.381,E2 -16831.381} C_VEL
LIN {X 0,Y 291.749,Z 609.143,A -85,B 0,C 180,E1 -16836.919,E2 -16836.919} C_VEL
LIN {X 0,Y 291.631,Z 609.155,A -85,B 0,C 180,E1 -16839.713,E2 -16839.713} C_VEL
LIN {X 0,Y 291.525,Z 609.168,A -85,B 0,C 180,E1 -16843.952,E2 -16843.952} C_VEL
LIN {X 0,Y 291.49,Z 609.177,A -85,B 0,C 180,E1 -16846.819,E2 -16846.819} C_VEL
LIN {X 0,Y 291.453,Z 609.173,A -85,B 0,C 180,E1 -16849.876,E2 -16849.876} C_VEL
LIN {X 0,Y 291.403,Z 609.183,A -85,B 0,C 180,E1 -16854.206,E2 -16854.206} C_VEL
LIN {X 0,Y 291.422,Z 609.184,A -85,B 0,C 180,E1 -16857.273,E2 -16857.273} C_VEL
LIN {X 0,Y 291.338,Z 609.191,A -85,B 0,C 180,E1 -16860.438,E2 -16860.438} C_VEL
LIN {X 0,Y 291.348,Z 609.185,A -85,B 0,C 180,E1 -16863.699,E2 -16863.699} C_VEL
LIN {X 0,Y 291.376,Z 609.189,A -85,B 0,C 180,E1 -16867.254,E2 -16867.254} C_VEL
LIN {X 0,Y 291.337,Z 609.192,A -85,B 0,C 180,E1 -16870.643,E2 -16870.643} C_VEL
LIN {X 0,Y 291.318,Z 609.193,A -85,B 0,C 180,E1 -16874.398,E2 -16874.398} C_VEL
LIN {X 0,Y 291.331,Z 609.189,A -85,B 0,C 180,E1 -16878.405,E2 -16878.405} C_VEL
LIN {X 0,Y 291.358,Z 609.186,A -85,B 0,C 180,E1 -16881.159,E2 -16881.159} C_VEL
LIN {X 0,Y 291.366,Z 609.183,A -85,B 0,C 180,E1 -16884.627,E2 -16884.627} C_VEL
LIN {X 0,Y 291.378,Z 609.188,A -85,B 0,C 180,E1 -16887.952,E2 -16887.952} C_VEL
LIN {X 0,Y 291.388,Z 609.186,A -85,B 0,C 180,E1 -16891.159,E2 -16891.159} C_VEL
LIN {X 0,Y 291.417,Z 609.181,A -85,B 0,C 180,E1 -16893.899,E2 -16893.899} C_VEL
LIN {X 0,Y 290.76,Z 609.266,A -85,B 0,C 180,E1 -16895.051,E2 -16895.051} C_VEL
LIN {X 0,Y 287.94,Z 609.623,A -85,B 0,C 180,E1 -16896.928,E2 -16896.928} C_VEL
LIN {X 0,Y 285.532,Z 609.922,A -85,B 0,C 180,E1 -16898.452,E2 -16898.452} C_VEL
LIN {X 0,Y 284.482,Z 610.047,A -85,B 0,C 180,E1 -16899.632,E2 -16899.632} C_VEL
LIN {X 0,Y 284.387,Z 610.056,A -85,B 0,C 180,E1 -16900.032,E2 -16900.032} C_VEL
LIN {X 0,Y 284.484,Z 610.039,A -85,B 0,C 180,E1 -16904.47,E2 -16904.47} C_VEL
LIN {X 0,Y 284.494,Z 610.043,A -85,B 0,C 180,E1 -16908.602,E2 -16908.602} C_VEL
LIN {X 0,Y 284.645,Z 610.026,A -85,B 0,C 180,E1 -16911.481,E2 -16911.481} C_VEL
LIN {X 0,Y 284.603,Z 610.033,A -85,B 0,C 180,E1 -16914.331,E2 -16914.331} C_VEL
LIN {X 0,Y 284.861,Z 609.997,A -85,B 0,C 180,E1 -16918.586,E2 -16918.586} C_VEL
LIN {X 0,Y 284.861,Z 609.993,A -85,B 0,C 180,E1 -16921.414,E2 -16921.414} C_VEL
LIN {X 0,Y 284.694,Z 610.019,A -85,B 0,C 180,E1 -16927.09,E2 -16927.09} C_VEL
LIN {X 0,Y 284.526,Z 610.042,A -85,B 0,C 180,E1 -16929.957,E2 -16929.957} C_VEL
LIN {X 0,Y 284.47,Z 610.049,A -85,B 0,C 180,E1 -16934.304,E2 -16934.304} C_VEL
LIN {X 0,Y 284.347,Z 610.066,A -85,B 0,C 180,E1 -16938.743,E2 -16938.743} C_VEL
LIN {X 0,Y 284.319,Z 610.067,A -85,B 0,C 180,E1 -16941.764,E2 -16941.764} C_VEL
LIN {X 0,Y 284.346,Z 610.065,A -85,B 0,C 180,E1 -16944.846,E2 -16944.846} C_VEL
LIN {X 0,Y 284.341,Z 610.064,A -85,B 0,C 180,E1 -16948.01,E2 -16948.01} C_VEL
LIN {X 0,Y 284.302,Z 610.069,A -85,B 0,C 180,E1 -16951.274,E2 -16951.274} C_VEL
LIN {X 0,Y 284.347,Z 610.064,A -85,B 0,C 180,E1 -16955.347,E2 -16955.347} C_VEL
LIN {X 0,Y 284.314,Z 610.067,A -85,B 0,C 180,E1 -16958.169,E2 -16958.169} C_VEL
LIN {X 0,Y 284.275,Z 610.072,A -85,B 0,C 180,E1 -16962.124,E2 -16962.124} C_VEL
LIN {X 0,Y 284.274,Z 610.072,A -85,B 0,C 180,E1 -16966.191,E2 -16966.191} C_VEL
LIN {X 0,Y 284.312,Z 610.068,A -85,B 0,C 180,E1 -16970.023,E2 -16970.023} C_VEL
LIN {X 0,Y 284.336,Z 610.068,A -85,B 0,C 180,E1 -16973.613,E2 -16973.613} C_VEL
LIN {X 0,Y 284.371,Z 610.254,A -85,B 0,C 180,E1 -16975.007,E2 -16975.007} C_VEL
LIN {X 0,Y 287.084,Z 623.086,A -85,B 0,C 180,E1 -16979.062,E2 -16979.062} C_VEL
LIN {X 0,Y 289.205,Z 633.292,A -85,B 0,C 180,E1 -16982.137,E2 -16982.137} C_VEL
LIN {X 0,Y 289.005,Z 637.328,A -85,B 0,C 180,E1 -16983.263,E2 -16983.263} C_VEL
LIN {X 0,Y 288.79,Z 638.761,A -85,B 0,C 180,E1 -16983.62,E2 -16983.62} C_VEL
LIN {X 0,Y 294.616,Z 686.264,A -85,B 0,C 180,E1 -16985.487,E2 -16985.487} C_VEL
LIN {X 0,Y 292.642,Z 747.995,A -85,B 0,C 180,E1 -16987.261,E2 -16987.261} C_VEL
LIN {X 0,Y 291.771,Z 761.804,A -85,B 0,C 180,E1 -16987.936,E2 -16987.936} C_VEL
LIN {X 0,Y 290.565,Z 774.289,A -85,B 0,C 180,E1 -16988.819,E2 -16988.819} C_VEL
LIN {X 0,Y 289.255,Z 785.936,A -85,B 0,C 180,E1 -16989.927,E2 -16989.927} C_VEL
LIN {X 0,Y 287.869,Z 797.295,A -85,B 0,C 180,E1 -16991.309,E2 -16991.309} C_VEL
LIN {X 0,Y 286.545,Z 807.576,A -85,B 0,C 180,E1 -16992.882,E2 -16992.882} C_VEL
LIN {X 0,Y 285.407,Z 816.857,A -85,B 0,C 180,E1 -16994.649,E2 -16994.649} C_VEL
LIN {X 0,Y 284.233,Z 825.888,A -85,B 0,C 180,E1 -16996.777,E2 -16996.777} C_VEL
LIN {X 0,Y 283.341,Z 833.077,A -85,B 0,C 180,E1 -16998.915,E2 -16998.915} C_VEL
LIN {X 0,Y 282.828,Z 839.629,A -85,B 0,C 180,E1 -17001.424,E2 -17001.424} C_VEL
LIN {X 0,Y 282.609,Z 843.889,A -85,B 0,C 180,E1 -17003.574,E2 -17003.574} C_VEL
LIN {X 0,Y 282.572,Z 847.014,A -85,B 0,C 180,E1 -17005.719,E2 -17005.719} C_VEL
LIN {X 0,Y 282.537,Z 848.529,A -85,B 0,C 180,E1 -17007.147,E2 -17007.147} C_VEL
LIN {X 0,Y 282.596,Z 849.564,A -85,B 0,C 180,E1 -17008.573,E2 -17008.573} C_VEL
LIN {X 0,Y 282.694,Z 850.178,A -85,B 0,C 180,E1 -17009.998,E2 -17009.998} C_VEL
LIN {X 0,Y 282.548,Z 850.363,A -85,B 0,C 180,E1 -17011.424,E2 -17011.424} C_VEL
LIN {X 0,Y 282.496,Z 850.129,A -85,B 0,C 180,E1 -17012.85,E2 -17012.85} C_VEL
LIN {X 0,Y 282.424,Z 848.534,A -85,B 0,C 180,E1 -17015.505,E2 -17015.505} C_VEL
LIN {X 0,Y 282.569,Z 846.852,A -85,B 0,C 180,E1 -17017.142,E2 -17017.142} C_VEL
LIN {X 0,Y 282.919,Z 843.748,A -85,B 0,C 180,E1 -17019.29,E2 -17019.29} C_VEL
LIN {X 0,Y 283.553,Z 839.611,A -85,B 0,C 180,E1 -17021.435,E2 -17021.435} C_VEL
LIN {X 0,Y 284.61,Z 834.334,A -85,B 0,C 180,E1 -17023.566,E2 -17023.566} C_VEL
LIN {X 0,Y 286.035,Z 827.757,A -85,B 0,C 180,E1 -17025.679,E2 -17025.679} C_VEL
LIN {X 0,Y 287.708,Z 819.919,A -85,B 0,C 180,E1 -17027.696,E2 -17027.696} C_VEL
LIN {X 0,Y 289.501,Z 811.314,A -85,B 0,C 180,E1 -17029.498,E2 -17029.498} C_VEL
LIN {X 0,Y 291.874,Z 800.244,A -85,B 0,C 180,E1 -17031.356,E2 -17031.356} C_VEL
LIN {X 0,Y 293.847,Z 790.297,A -85,B 0,C 180,E1 -17032.683,E2 -17032.683} C_VEL
LIN {X 0,Y 295.72,Z 779.643,A -85,B 0,C 180,E1 -17033.828,E2 -17033.828} C_VEL
LIN {X 0,Y 297.689,Z 767.057,A -85,B 0,C 180,E1 -17034.866,E2 -17034.866} C_VEL
LIN {X 0,Y 299.174,Z 754.782,A -85,B 0,C 180,E1 -17035.617,E2 -17035.617} C_VEL
LIN {X 0,Y 300.234,Z 741.393,A -85,B 0,C 180,E1 -17036.172,E2 -17036.172} C_VEL
LIN {X 0,Y 302.768,Z 686.931,A -85,B 0,C 180,E1 -17037.773,E2 -17037.773} C_VEL
LIN {X 0,Y 300.809,Z 669.044,A -85,B 0,C 180,E1 -17038.701,E2 -17038.701} C_VEL
LIN {X 0,Y 297.795,Z 651.591,A -85,B 0,C 180,E1 -17039.799,E2 -17039.799} C_VEL
LIN {X 0,Y 296.681,Z 647.232,A -85,B 0,C 180,E1 -17040.139,E2 -17040.139} C_VEL
LIN {X 0,Y 292.212,Z 637.685,A -85,B 0,C 180,E1 -17041.25,E2 -17041.25} C_VEL
LIN {X 0,Y 290.464,Z 633.815,A -85,B 0,C 180,E1 -17041.747,E2 -17041.747} C_VEL
LIN {X 0,Y 288.678,Z 625.725,A -85,B 0,C 180,E1 -17044.895,E2 -17044.895} C_VEL
LIN {X 0,Y 286.592,Z 617.894,A -85,B 0,C 180,E1 -17048.304,E2 -17048.304} C_VEL
LIN {X 0,Y 284.918,Z 612.116,A -85,B 0,C 180,E1 -17051.13,E2 -17051.13} C_VEL
LIN {X 0,Y 284.337,Z 610.07,A -85,B 0,C 180,E1 -17052.234,E2 -17052.234} C_VEL
LIN {X 0,Y 284.326,Z 610.069,A -85,B 0,C 180,E1 -17056.203,E2 -17056.203} C_VEL
LIN {X 0,Y 284.346,Z 610.068,A -85,B 0,C 180,E1 -17060.012,E2 -17060.012} C_VEL
LIN {X 0,Y 284.35,Z 610.06,A -85,B 0,C 180,E1 -17063.616,E2 -17063.616} C_VEL
LIN {X 0,Y 284.303,Z 610.07,A -85,B 0,C 180,E1 -17067.188,E2 -17067.188} C_VEL
LIN {X 0,Y 284.353,Z 610.06,A -85,B 0,C 180,E1 -17070.375,E2 -17070.375} C_VEL
LIN {X 0,Y 284.371,Z 610.055,A -85,B 0,C 180,E1 -17073.586,E2 -17073.586} C_VEL
LIN {X 0,Y 284.361,Z 610.057,A -85,B 0,C 180,E1 -17076.706,E2 -17076.706} C_VEL
LIN {X 0,Y 284.396,Z 610.06,A -85,B 0,C 180,E1 -17081.261,E2 -17081.261} C_VEL
LIN {X 0,Y 284.484,Z 610.046,A -85,B 0,C 180,E1 -17084.458,E2 -17084.458} C_VEL
LIN {X 0,Y 284.482,Z 610.048,A -85,B 0,C 180,E1 -17088.601,E2 -17088.601} C_VEL
LIN {X 0,Y 284.651,Z 610.029,A -85,B 0,C 180,E1 -17091.481,E2 -17091.481} C_VEL
LIN {X 0,Y 284.594,Z 610.034,A -85,B 0,C 180,E1 -17094.331,E2 -17094.331} C_VEL
LIN {X 0,Y 284.849,Z 610.002,A -85,B 0,C 180,E1 -17098.586,E2 -17098.586} C_VEL
LIN {X 0,Y 284.865,Z 610.015,A -85,B 0,C 180,E1 -17101.06,E2 -17101.06} C_VEL
LIN {X 0,Y 285.45,Z 612.578,A -85,B 0,C 180,E1 -17102.469,E2 -17102.469} C_VEL
LIN {X 0,Y 287.5,Z 616.207,A -85,B 0,C 180,E1 -17103.021,E2 -17103.021} C_VEL
LIN {X 0,Y 295.225,Z 628.754,A -85,B 0,C 180,E1 -17104.9,E2 -17104.9} C_VEL
LIN {X 0,Y 300.895,Z 640.155,A -85,B 0,C 180,E1 -17106.235,E2 -17106.235} C_VEL
LIN {X 0,Y 304.404,Z 648.165,A -85,B 0,C 180,E1 -17107.043,E2 -17107.043} C_VEL
LIN {X 0,Y 300.946,Z 717.526,A -85,B 0,C 180,E1 -17109.119,E2 -17109.119} C_VEL
LIN {X 0,Y 299.86,Z 730.885,A -85,B 0,C 180,E1 -17109.777,E2 -17109.777} C_VEL
LIN {X 0,Y 298.547,Z 743.651,A -85,B 0,C 180,E1 -17110.7,E2 -17110.7} C_VEL
LIN {X 0,Y 296.969,Z 754.923,A -85,B 0,C 180,E1 -17111.778,E2 -17111.778} C_VEL
LIN {X 0,Y 295.285,Z 765.137,A -85,B 0,C 180,E1 -17113.012,E2 -17113.012} C_VEL
LIN {X 0,Y 293.276,Z 775.555,A -85,B 0,C 180,E1 -17114.573,E2 -17114.573} C_VEL
LIN {X 0,Y 291.374,Z 784.156,A -85,B 0,C 180,E1 -17116.167,E2 -17116.167} C_VEL
LIN {X 0,Y 289.482,Z 792.277,A -85,B 0,C 180,E1 -17118.031,E2 -17118.031} C_VEL
LIN {X 0,Y 287.464,Z 800.298,A -85,B 0,C 180,E1 -17120.336,E2 -17120.336} C_VEL
LIN {X 0,Y 286.094,Z 805.845,A -85,B 0,C 180,E1 -17122.381,E2 -17122.381} C_VEL
LIN {X 0,Y 284.821,Z 810.864,A -85,B 0,C 180,E1 -17124.801,E2 -17124.801} C_VEL
LIN {X 0,Y 283.91,Z 814.173,A -85,B 0,C 180,E1 -17126.985,E2 -17126.985} C_VEL
LIN {X 0,Y 283.072,Z 816.869,A -85,B 0,C 180,E1 -17129.772,E2 -17129.772} C_VEL
LIN {X 0,Y 282.623,Z 817.945,A -85,B 0,C 180,E1 -17132.28,E2 -17132.28} C_VEL
LIN {X 0,Y 282.427,Z 817.67,A -85,B 0,C 180,E1 -17134.913,E2 -17134.913} C_VEL
LIN {X 0,Y 282.433,Z 816.284,A -85,B 0,C 180,E1 -17137.227,E2 -17137.227} C_VEL
LIN {X 0,Y 282.671,Z 813.727,A -85,B 0,C 180,E1 -17139.582,E2 -17139.582} C_VEL
LIN {X 0,Y 283.155,Z 809.683,A -85,B 0,C 180,E1 -17142.078,E2 -17142.078} C_VEL
LIN {X 0,Y 283.751,Z 804.468,A -85,B 0,C 180,E1 -17144.426,E2 -17144.426} C_VEL
LIN {X 0,Y 284.523,Z 798.495,A -85,B 0,C 180,E1 -17146.514,E2 -17146.514} C_VEL
LIN {X 0,Y 285.47,Z 791.179,A -85,B 0,C 180,E1 -17148.569,E2 -17148.569} C_VEL
LIN {X 0,Y 286.715,Z 782.376,A -85,B 0,C 180,E1 -17150.563,E2 -17150.563} C_VEL
LIN {X 0,Y 288.061,Z 772.124,A -85,B 0,C 180,E1 -17152.417,E2 -17152.417} C_VEL
LIN {X 0,Y 289.494,Z 760.637,A -85,B 0,C 180,E1 -17154.071,E2 -17154.071} C_VEL
LIN {X 0,Y 290.685,Z 748.611,A -85,B 0,C 180,E1 -17155.427,E2 -17155.427} C_VEL
LIN {X 0,Y 291.81,Z 736.479,A -85,B 0,C 180,E1 -17156.475,E2 -17156.475} C_VEL
LIN {X 0,Y 292.638,Z 723.222,A -85,B 0,C 180,E1 -17157.318,E2 -17157.318} C_VEL
LIN {X 0,Y 293.259,Z 709.308,A -85,B 0,C 180,E1 -17157.887,E2 -17157.887} C_VEL
LIN {X 0,Y 295.462,Z 639.698,A -85,B 0,C 180,E1 -17159.849,E2 -17159.849} C_VEL
LIN {X 0,Y 288.86,Z 621.458,A -85,B 0,C 180,E1 -17160.884,E2 -17160.884} C_VEL
LIN {X 0,Y 284.483,Z 610.754,A -85,B 0,C 180,E1 -17161.556,E2 -17161.556} C_VEL
LIN {X 0,Y 284.334,Z 610.067,A -85,B 0,C 180,E1 -17161.59,E2 -17161.59} C_VEL
LIN {X 0,Y 284.343,Z 610.063,A -85,B 0,C 180,E1 -17165.156,E2 -17165.156} C_VEL
LIN {X 0,Y 284.337,Z 610.069,A -85,B 0,C 180,E1 -17168.239,E2 -17168.239} C_VEL
LIN {X 0,Y 284.404,Z 610.056,A -85,B 0,C 180,E1 -17171.263,E2 -17171.263} C_VEL
LIN {X 0,Y 284.491,Z 610.048,A -85,B 0,C 180,E1 -17174.461,E2 -17174.461} C_VEL
LIN {X 0,Y 284.489,Z 610.048,A -85,B 0,C 180,E1 -17178.603,E2 -17178.603} C_VEL
LIN {X 0,Y 284.659,Z 610.024,A -85,B 0,C 180,E1 -17181.483,E2 -17181.483} C_VEL
LIN {X 0,Y 284.602,Z 610.036,A -85,B 0,C 180,E1 -17184.333,E2 -17184.333} C_VEL
LIN {X 0,Y 284.856,Z 610.004,A -85,B 0,C 180,E1 -17188.588,E2 -17188.588} C_VEL
LIN {X 0,Y 284.86,Z 609.999,A -85,B 0,C 180,E1 -17191.415,E2 -17191.415} C_VEL
LIN {X 0,Y 284.701,Z 610.02,A -85,B 0,C 180,E1 -17197.091,E2 -17197.091} C_VEL
LIN {X 0,Y 284.569,Z 610.035,A -85,B 0,C 180,E1 -17199.957,E2 -17199.957} C_VEL
LIN {X 0,Y 284.484,Z 610.047,A -85,B 0,C 180,E1 -17204.304,E2 -17204.304} C_VEL
LIN {X 0,Y 284.428,Z 610.052,A -85,B 0,C 180,E1 -17207.25,E2 -17207.25} C_VEL
LIN {X 0,Y 284.381,Z 610.054,A -85,B 0,C 180,E1 -17210.243,E2 -17210.243} C_VEL
LIN {X 0,Y 284.372,Z 610.059,A -85,B 0,C 180,E1 -17213.877,E2 -17213.877} C_VEL
LIN {X 0,Y 284.398,Z 610.06,A -85,B 0,C 180,E1 -17217.174,E2 -17217.174} C_VEL
LIN {X 0,Y 284.297,Z 610.068,A -85,B 0,C 180,E1 -17221.276,E2 -17221.276} C_VEL
LIN {X 0,Y 284.345,Z 610.063,A -85,B 0,C 180,E1 -17225.349,E2 -17225.349} C_VEL
LIN {X 0,Y 284.312,Z 610.065,A -85,B 0,C 180,E1 -17228.171,E2 -17228.171} C_VEL
LIN {X 0,Y 284.274,Z 610.071,A -85,B 0,C 180,E1 -17232.125,E2 -17232.125} C_VEL
LIN {X 0,Y 284.273,Z 610.07,A -85,B 0,C 180,E1 -17236.193,E2 -17236.193} C_VEL
LIN {X 0,Y 284.311,Z 610.062,A -85,B 0,C 180,E1 -17240.025,E2 -17240.025} C_VEL
LIN {X 0,Y 284.337,Z 610.061,A -85,B 0,C 180,E1 -17243.615,E2 -17243.615} C_VEL
LIN {X 0,Y 284.313,Z 610.065,A -85,B 0,C 180,E1 -17247.19,E2 -17247.19} C_VEL
LIN {X 0,Y 284.364,Z 610.06,A -85,B 0,C 180,E1 -17250.377,E2 -17250.377} C_VEL
LIN {X 0,Y 284.36,Z 610.063,A -85,B 0,C 180,E1 -17253.88,E2 -17253.88} C_VEL
LIN {X 0,Y 284.339,Z 610.062,A -85,B 0,C 180,E1 -17256.705,E2 -17256.705} C_VEL
LIN {X 0,Y 284.387,Z 610.056,A -85,B 0,C 180,E1 -17260.032,E2 -17260.032} C_VEL
LIN {X 0,Y 283.699,Z 610.141,A -85,B 0,C 180,E1 -17261.216,E2 -17261.216} C_VEL
LIN {X 0,Y 280.864,Z 610.488,A -85,B 0,C 180,E1 -17263.145,E2 -17263.145} C_VEL
LIN {X 0,Y 278.485,Z 610.785,A -85,B 0,C 180,E1 -17264.711,E2 -17264.711} C_VEL
LIN {X 0,Y 277.48,Z 610.915,A -85,B 0,C 180,E1 -17265.924,E2 -17265.924} C_VEL
LIN {X 0,Y 277.405,Z 610.919,A -85,B 0,C 180,E1 -17266.335,E2 -17266.335} C_VEL
LIN {X 0,Y 277.576,Z 610.905,A -85,B 0,C 180,E1 -17270.92,E2 -17270.92} C_VEL
LIN {X 0,Y 277.573,Z 610.91,A -85,B 0,C 180,E1 -17274.187,E2 -17274.187} C_VEL
LIN {X 0,Y 277.827,Z 610.873,A -85,B 0,C 180,E1 -17278.551,E2 -17278.551} C_VEL
LIN {X 0,Y 277.827,Z 610.868,A -85,B 0,C 180,E1 -17281.45,E2 -17281.45} C_VEL
LIN {X 0,Y 277.648,Z 610.897,A -85,B 0,C 180,E1 -17287.271,E2 -17287.271} C_VEL
LIN {X 0,Y 277.468,Z 610.923,A -85,B 0,C 180,E1 -17290.213,E2 -17290.213} C_VEL
LIN {X 0,Y 277.416,Z 610.925,A -85,B 0,C 180,E1 -17294.675,E2 -17294.675} C_VEL
LIN {X 0,Y 277.311,Z 610.94,A -85,B 0,C 180,E1 -17299.237,E2 -17299.237} C_VEL
LIN {X 0,Y 277.304,Z 610.94,A -85,B 0,C 180,E1 -17303.923,E2 -17303.923} C_VEL
LIN {X 0,Y 277.334,Z 610.937,A -85,B 0,C 180,E1 -17307.506,E2 -17307.506} C_VEL
LIN {X 0,Y 277.278,Z 610.947,A -85,B 0,C 180,E1 -17310.481,E2 -17310.481} C_VEL
LIN {X 0,Y 277.253,Z 610.946,A -85,B 0,C 180,E1 -17313.895,E2 -17313.895} C_VEL
LIN {X 0,Y 277.271,Z 610.945,A -85,B 0,C 180,E1 -17317.469,E2 -17317.469} C_VEL
LIN {X 0,Y 277.216,Z 610.955,A -85,B 0,C 180,E1 -17321.236,E2 -17321.236} C_VEL
LIN {X 0,Y 277.222,Z 610.954,A -85,B 0,C 180,E1 -17325.222,E2 -17325.222} C_VEL
LIN {X 0,Y 277.228,Z 610.952,A -85,B 0,C 180,E1 -17329.511,E2 -17329.511} C_VEL
LIN {X 0,Y 277.27,Z 610.946,A -85,B 0,C 180,E1 -17332.529,E2 -17332.529} C_VEL
LIN {X 0,Y 277.318,Z 611.013,A -85,B 0,C 180,E1 -17334.568,E2 -17334.568} C_VEL
LIN {X 0,Y 279.937,Z 623.438,A -85,B 0,C 180,E1 -17338.605,E2 -17338.605} C_VEL
LIN {X 0,Y 282.283,Z 634.984,A -85,B 0,C 180,E1 -17342.171,E2 -17342.171} C_VEL
LIN {X 0,Y 282.003,Z 638.24,A -85,B 0,C 180,E1 -17343.096,E2 -17343.096} C_VEL
LIN {X 0,Y 287.846,Z 686.932,A -85,B 0,C 180,E1 -17345.072,E2 -17345.072} C_VEL
LIN {X 0,Y 285.812,Z 747.944,A -85,B 0,C 180,E1 -17346.878,E2 -17346.878} C_VEL
LIN {X 0,Y 284.912,Z 761.623,A -85,B 0,C 180,E1 -17347.567,E2 -17347.567} C_VEL
LIN {X 0,Y 283.685,Z 774.033,A -85,B 0,C 180,E1 -17348.47,E2 -17348.47} C_VEL
LIN {X 0,Y 282.366,Z 785.656,A -85,B 0,C 180,E1 -17349.606,E2 -17349.606} C_VEL
LIN {X 0,Y 280.933,Z 796.991,A -85,B 0,C 180,E1 -17351.02,E2 -17351.02} C_VEL
LIN {X 0,Y 279.512,Z 807.673,A -85,B 0,C 180,E1 -17352.706,E2 -17352.706} C_VEL
LIN {X 0,Y 278.266,Z 817.349,A -85,B 0,C 180,E1 -17354.62,E2 -17354.62} C_VEL
LIN {X 0,Y 277.108,Z 826.207,A -85,B 0,C 180,E1 -17356.804,E2 -17356.804} C_VEL
LIN {X 0,Y 276.222,Z 833.236,A -85,B 0,C 180,E1 -17358.998,E2 -17358.998} C_VEL
LIN {X 0,Y 275.774,Z 838.847,A -85,B 0,C 180,E1 -17361.203,E2 -17361.203} C_VEL
LIN {X 0,Y 275.542,Z 843.194,A -85,B 0,C 180,E1 -17363.408,E2 -17363.408} C_VEL
LIN {X 0,Y 275.488,Z 846.398,A -85,B 0,C 180,E1 -17365.609,E2 -17365.609} C_VEL
LIN {X 0,Y 275.464,Z 847.959,A -85,B 0,C 180,E1 -17367.074,E2 -17367.074} C_VEL
LIN {X 0,Y 275.508,Z 849.056,A -85,B 0,C 180,E1 -17368.537,E2 -17368.537} C_VEL
LIN {X 0,Y 275.607,Z 849.704,A -85,B 0,C 180,E1 -17369.998,E2 -17369.998} C_VEL
LIN {X 0,Y 275.462,Z 849.922,A -85,B 0,C 180,E1 -17371.46,E2 -17371.46} C_VEL
LIN {X 0,Y 275.418,Z 849.735,A -85,B 0,C 180,E1 -17372.924,E2 -17372.924} C_VEL
LIN {X 0,Y 275.35,Z 848.37,A -85,B 0,C 180,E1 -17375.476,E2 -17375.476} C_VEL
LIN {X 0,Y 275.498,Z 846.58,A -85,B 0,C 180,E1 -17377.326,E2 -17377.326} C_VEL
LIN {X 0,Y 275.889,Z 843.56,A -85,B 0,C 180,E1 -17379.529,E2 -17379.529} C_VEL
LIN {X 0,Y 276.543,Z 839.498,A -85,B 0,C 180,E1 -17381.729,E2 -17381.729} C_VEL
LIN {X 0,Y 277.923,Z 833.336,A -85,B 0,C 180,E1 -17384.272,E2 -17384.272} C_VEL
LIN {X 0,Y 279.432,Z 826.588,A -85,B 0,C 180,E1 -17386.435,E2 -17386.435} C_VEL
LIN {X 0,Y 281.251,Z 818.75,A -85,B 0,C 180,E1 -17388.467,E2 -17388.467} C_VEL
LIN {X 0,Y 283.298,Z 809.925,A -85,B 0,C 180,E1 -17390.321,E2 -17390.321} C_VEL
LIN {X 0,Y 285.535,Z 799.774,A -85,B 0,C 180,E1 -17392.044,E2 -17392.044} C_VEL
LIN {X 0,Y 287.886,Z 788.402,A -85,B 0,C 180,E1 -17393.561,E2 -17393.561} C_VEL
LIN {X 0,Y 289.908,Z 777.418,A -85,B 0,C 180,E1 -17394.718,E2 -17394.718} C_VEL
LIN {X 0,Y 291.815,Z 765.471,A -85,B 0,C 180,E1 -17395.689,E2 -17395.689} C_VEL
LIN {X 0,Y 293.475,Z 751.892,A -85,B 0,C 180,E1 -17396.487,E2 -17396.487} C_VEL
LIN {X 0,Y 294.475,Z 738.657,A -85,B 0,C 180,E1 -17397.016,E2 -17397.016} C_VEL
LIN {X 0,Y 296.999,Z 687.969,A -85,B 0,C 180,E1 -17398.537,E2 -17398.537} C_VEL
LIN {X 0,Y 295.111,Z 670.337,A -85,B 0,C 180,E1 -17399.485,E2 -17399.485} C_VEL
LIN {X 0,Y 292.164,Z 652.761,A -85,B 0,C 180,E1 -17400.647,E2 -17400.647} C_VEL
LIN {X 0,Y 291.198,Z 649.966,A -85,B 0,C 180,E1 -17400.92,E2 -17400.92} C_VEL
LIN {X 0,Y 287.442,Z 641.868,A -85,B 0,C 180,E1 -17401.896,E2 -17401.896} C_VEL
LIN {X 0,Y 283.23,Z 633.18,A -85,B 0,C 180,E1 -17403.084,E2 -17403.084} C_VEL
LIN {X 0,Y 281.374,Z 625.124,A -85,B 0,C 180,E1 -17406.456,E2 -17406.456} C_VEL
LIN {X 0,Y 279.388,Z 617.855,A -85,B 0,C 180,E1 -17409.894,E2 -17409.894} C_VEL
LIN {X 0,Y 277.3,Z 610.948,A -85,B 0,C 180,E1 -17413.736,E2 -17413.736} C_VEL
LIN {X 0,Y 277.27,Z 610.948,A -85,B 0,C 180,E1 -17417.31,E2 -17417.31} C_VEL
LIN {X 0,Y 277.263,Z 610.945,A -85,B 0,C 180,E1 -17420.676,E2 -17420.676} C_VEL
LIN {X 0,Y 277.3,Z 610.941,A -85,B 0,C 180,E1 -17424.343,E2 -17424.343} C_VEL
LIN {X 0,Y 277.24,Z 610.947,A -85,B 0,C 180,E1 -17427.835,E2 -17427.835} C_VEL
LIN {X 0,Y 277.265,Z 610.938,A -85,B 0,C 180,E1 -17431.209,E2 -17431.209} C_VEL
LIN {X 0,Y 277.307,Z 610.935,A -85,B 0,C 180,E1 -17434.479,E2 -17434.479} C_VEL
LIN {X 0,Y 277.284,Z 610.942,A -85,B 0,C 180,E1 -17437.654,E2 -17437.654} C_VEL
LIN {X 0,Y 277.338,Z 610.939,A -85,B 0,C 180,E1 -17440.765,E2 -17440.765} C_VEL
LIN {X 0,Y 277.427,Z 610.922,A -85,B 0,C 180,E1 -17445.325,E2 -17445.325} C_VEL
LIN {X 0,Y 277.499,Z 610.916,A -85,B 0,C 180,E1 -17449.788,E2 -17449.788} C_VEL
LIN {X 0,Y 277.645,Z 610.897,A -85,B 0,C 180,E1 -17452.729,E2 -17452.729} C_VEL
LIN {X 0,Y 277.815,Z 610.878,A -85,B 0,C 180,E1 -17458.55,E2 -17458.55} C_VEL
LIN {X 0,Y 277.859,Z 610.897,A -85,B 0,C 180,E1 -17459.637,E2 -17459.637} C_VEL
LIN {X 0,Y 278.519,Z 613.323,A -85,B 0,C 180,E1 -17461.084,E2 -17461.084} C_VEL
LIN {X 0,Y 280.58,Z 616.817,A -85,B 0,C 180,E1 -17461.687,E2 -17461.687} C_VEL
LIN {X 0,Y 281.822,Z 618.769,A -85,B 0,C 180,E1 -17462.033,E2 -17462.033} C_VEL
LIN {X 0,Y 290.457,Z 632.856,A -85,B 0,C 180,E1 -17464.265,E2 -17464.265} C_VEL
LIN {X 0,Y 296.367,Z 645.104,A -85,B 0,C 180,E1 -17465.741,E2 -17465.741} C_VEL
LIN {X 0,Y 298.623,Z 650.292,A -85,B 0,C 180,E1 -17466.283,E2 -17466.283} C_VEL
LIN {X 0,Y 295.105,Z 717.688,A -85,B 0,C 180,E1 -17468.344,E2 -17468.344} C_VEL
LIN {X 0,Y 293.951,Z 731.27,A -85,B 0,C 180,E1 -17469.027,E2 -17469.027} C_VEL
LIN {X 0,Y 292.55,Z 743.983,A -85,B 0,C 180,E1 -17469.963,E2 -17469.963} C_VEL
LIN {X 0,Y 290.767,Z 756.015,A -85,B 0,C 180,E1 -17471.149,E2 -17471.149} C_VEL
LIN {X 0,Y 288.894,Z 766.605,A -85,B 0,C 180,E1 -17472.468,E2 -17472.468} C_VEL
LIN {X 0,Y 286.624,Z 777.566,A -85,B 0,C 180,E1 -17474.193,E2 -17474.193} C_VEL
LIN {X 0,Y 284.72,Z 785.594,A -85,B 0,C 180,E1 -17475.755,E2 -17475.755} C_VEL
LIN {X 0,Y 282.754,Z 793.547,A -85,B 0,C 180,E1 -17477.66,E2 -17477.66} C_VEL
LIN {X 0,Y 280.886,Z 800.545,A -85,B 0,C 180,E1 -17479.742,E2 -17479.742} C_VEL
LIN {X 0,Y 279.135,Z 806.948,A -85,B 0,C 180,E1 -17482.189,E2 -17482.189} C_VEL
LIN {X 0,Y 277.916,Z 811.426,A -85,B 0,C 180,E1 -17484.447,E2 -17484.447} C_VEL
LIN {X 0,Y 276.752,Z 815.308,A -85,B 0,C 180,E1 -17487.2,E2 -17487.2} C_VEL
LIN {X 0,Y 275.94,Z 817.644,A -85,B 0,C 180,E1 -17490.012,E2 -17490.012} C_VEL
LIN {X 0,Y 275.479,Z 818.424,A -85,B 0,C 180,E1 -17492.663,E2 -17492.663} C_VEL
LIN {X 0,Y 275.317,Z 817.911,A -85,B 0,C 180,E1 -17495.231,E2 -17495.231} C_VEL
LIN {X 0,Y 275.374,Z 816.166,A -85,B 0,C 180,E1 -17497.772,E2 -17497.772} C_VEL
LIN {X 0,Y 275.691,Z 813.391,A -85,B 0,C 180,E1 -17500.116,E2 -17500.116} C_VEL
LIN {X 0,Y 276.134,Z 809.473,A -85,B 0,C 180,E1 -17502.434,E2 -17502.434} C_VEL
LIN {X 0,Y 276.746,Z 804.438,A -85,B 0,C 180,E1 -17504.681,E2 -17504.681} C_VEL
LIN {X 0,Y 277.704,Z 797.098,A -85,B 0,C 180,E1 -17507.216,E2 -17507.216} C_VEL
LIN {X 0,Y 278.818,Z 788.981,A -85,B 0,C 180,E1 -17509.406,E2 -17509.406} C_VEL
LIN {X 0,Y 280.083,Z 780.132,A -85,B 0,C 180,E1 -17511.323,E2 -17511.323} C_VEL
LIN {X 0,Y 281.518,Z 769.433,A -85,B 0,C 180,E1 -17513.193,E2 -17513.193} C_VEL
LIN {X 0,Y 282.917,Z 758.073,A -85,B 0,C 180,E1 -17514.756,E2 -17514.756} C_VEL
LIN {X 0,Y 284.136,Z 746.378,A -85,B 0,C 180,E1 -17516.031,E2 -17516.031} C_VEL
LIN {X 0,Y 285.177,Z 734.11,A -85,B 0,C 180,E1 -17517.051,E2 -17517.051} C_VEL
LIN {X 0,Y 285.994,Z 720.097,A -85,B 0,C 180,E1 -17517.887,E2 -17517.887} C_VEL
LIN {X 0,Y 286.564,Z 705.698,A -85,B 0,C 180,E1 -17518.413,E2 -17518.413} C_VEL
LIN {X 0,Y 288.723,Z 641.073,A -85,B 0,C 180,E1 -17520.275,E2 -17520.275} C_VEL
LIN {X 0,Y 282.474,Z 623.949,A -85,B 0,C 180,E1 -17521.284,E2 -17521.284} C_VEL
LIN {X 0,Y 277.468,Z 611.759,A -85,B 0,C 180,E1 -17522.078,E2 -17522.078} C_VEL
LIN {X 0,Y 277.34,Z 610.94,A -85,B 0,C 180,E1 -17522.152,E2 -17522.152} C_VEL
LIN {X 0,Y 277.326,Z 610.942,A -85,B 0,C 180,E1 -17526.081,E2 -17526.081} C_VEL
LIN {X 0,Y 277.345,Z 610.936,A -85,B 0,C 180,E1 -17530.768,E2 -17530.768} C_VEL
LIN {X 0,Y 277.434,Z 610.924,A -85,B 0,C 180,E1 -17535.328,E2 -17535.328} C_VEL
LIN {X 0,Y 277.507,Z 610.916,A -85,B 0,C 180,E1 -17539.79,E2 -17539.79} C_VEL
LIN {X 0,Y 277.653,Z 610.9,A -85,B 0,C 180,E1 -17542.731,E2 -17542.731} C_VEL
LIN {X 0,Y 277.822,Z 610.88,A -85,B 0,C 180,E1 -17548.552,E2 -17548.552} C_VEL
LIN {X 0,Y 277.826,Z 610.875,A -85,B 0,C 180,E1 -17551.451,E2 -17551.451} C_VEL
LIN {X 0,Y 277.655,Z 610.897,A -85,B 0,C 180,E1 -17557.272,E2 -17557.272} C_VEL
LIN {X 0,Y 277.509,Z 610.916,A -85,B 0,C 180,E1 -17560.213,E2 -17560.213} C_VEL
LIN {X 0,Y 277.437,Z 610.927,A -85,B 0,C 180,E1 -17564.675,E2 -17564.675} C_VEL
LIN {X 0,Y 277.348,Z 610.931,A -85,B 0,C 180,E1 -17569.235,E2 -17569.235} C_VEL
LIN {X 0,Y 277.322,Z 610.937,A -85,B 0,C 180,E1 -17574.171,E2 -17574.171} C_VEL
LIN {X 0,Y 277.326,Z 610.938,A -85,B 0,C 180,E1 -17577.505,E2 -17577.505} C_VEL
LIN {X 0,Y 277.275,Z 610.942,A -85,B 0,C 180,E1 -17580.483,E2 -17580.483} C_VEL
LIN {X 0,Y 277.25,Z 610.938,A -85,B 0,C 180,E1 -17583.897,E2 -17583.897} C_VEL
LIN {X 0,Y 277.269,Z 610.945,A -85,B 0,C 180,E1 -17587.471,E2 -17587.471} C_VEL
LIN {X 0,Y 277.214,Z 610.955,A -85,B 0,C 180,E1 -17591.238,E2 -17591.238} C_VEL
LIN {X 0,Y 277.221,Z 610.953,A -85,B 0,C 180,E1 -17595.224,E2 -17595.224} C_VEL
LIN {X 0,Y 277.227,Z 610.947,A -85,B 0,C 180,E1 -17599.513,E2 -17599.513} C_VEL
LIN {X 0,Y 277.272,Z 610.932,A -85,B 0,C 180,E1 -17602.532,E2 -17602.532} C_VEL
LIN {X 0,Y 277.252,Z 610.943,A -85,B 0,C 180,E1 -17606.105,E2 -17606.105} C_VEL
LIN {X 0,Y 277.267,Z 610.947,A -85,B 0,C 180,E1 -17609.539,E2 -17609.539} C_VEL
LIN {X 0,Y 277.365,Z 610.932,A -85,B 0,C 180,E1 -17612.865,E2 -17612.865} C_VEL
LIN {X 0,Y 277.303,Z 610.941,A -85,B 0,C 180,E1 -17616.077,E2 -17616.077} C_VEL
LIN {X 0,Y 277.348,Z 610.928,A -85,B 0,C 180,E1 -17620.767,E2 -17620.767} C_VEL
LIN {X 0,Y 277.434,Z 610.916,A -85,B 0,C 180,E1 -17625.326,E2 -17625.326} C_VEL
LIN {X 0,Y 277.405,Z 610.919,A -85,B 0,C 180,E1 -17626.335,E2 -17626.335} C_VEL
LIN {X 0,Y 276.792,Z 611.002,A -85,B 0,C 180,E1 -17627.547,E2 -17627.547} C_VEL
LIN {X 0,Y 274.083,Z 611.344,A -85,B 0,C 180,E1 -17629.526,E2 -17629.526} C_VEL
LIN {X 0,Y 270.933,Z 611.737,A -85,B 0,C 180,E1 -17631.958,E2 -17631.958} C_VEL
LIN {X 0,Y 270.581,Z 611.777,A -85,B 0,C 180,E1 -17632.797,E2 -17632.797} C_VEL
LIN {X 0,Y 270.793,Z 611.749,A -85,B 0,C 180,E1 -17638.513,E2 -17638.513} C_VEL
LIN {X 0,Y 270.793,Z 611.743,A -85,B 0,C 180,E1 -17641.487,E2 -17641.487} C_VEL
LIN {X 0,Y 270.606,Z 611.774,A -85,B 0,C 180,E1 -17647.462,E2 -17647.462} C_VEL
LIN {X 0,Y 270.419,Z 611.801,A -85,B 0,C 180,E1 -17650.482,E2 -17650.482} C_VEL
LIN {X 0,Y 270.374,Z 611.8,A -85,B 0,C 180,E1 -17655.066,E2 -17655.066} C_VEL
LIN {X 0,Y 270.258,Z 611.819,A -85,B 0,C 180,E1 -17659.759,E2 -17659.759} C_VEL
LIN {X 0,Y 270.245,Z 611.822,A -85,B 0,C 180,E1 -17664.589,E2 -17664.589} C_VEL
LIN {X 0,Y 270.279,Z 611.816,A -85,B 0,C 180,E1 -17667.908,E2 -17667.908} C_VEL
LIN {X 0,Y 270.191,Z 611.827,A -85,B 0,C 180,E1 -17671.348,E2 -17671.348} C_VEL
LIN {X 0,Y 270.208,Z 611.829,A -85,B 0,C 180,E1 -17674.905,E2 -17674.905} C_VEL
LIN {X 0,Y 270.203,Z 611.828,A -85,B 0,C 180,E1 -17678.71,E2 -17678.71} C_VEL
LIN {X 0,Y 270.177,Z 611.832,A -85,B 0,C 180,E1 -17683.25,E2 -17683.25} C_VEL
LIN {X 0,Y 270.18,Z 611.83,A -85,B 0,C 180,E1 -17687.441,E2 -17687.441} C_VEL
LIN {X 0,Y 270.212,Z 611.828,A -85,B 0,C 180,E1 -17691.373,E2 -17691.373} C_VEL
LIN {X 0,Y 270.263,Z 611.988,A -85,B 0,C 180,E1 -17694.188,E2 -17694.188} C_VEL
LIN {X 0,Y 272.843,Z 624.034,A -85,B 0,C 180,E1 -17698.215,E2 -17698.215} C_VEL
LIN {X 0,Y 275.138,Z 635.318,A -85,B 0,C 180,E1 -17701.798,E2 -17701.798} C_VEL
LIN {X 0,Y 275.22,Z 637.875,A -85,B 0,C 180,E1 -17702.563,E2 -17702.563} C_VEL
LIN {X 0,Y 281.104,Z 687.23,A -85,B 0,C 180,E1 -17704.626,E2 -17704.626} C_VEL
LIN {X 0,Y 279.075,Z 746.862,A -85,B 0,C 180,E1 -17706.434,E2 -17706.434} C_VEL
LIN {X 0,Y 278.152,Z 760.728,A -85,B 0,C 180,E1 -17707.139,E2 -17707.139} C_VEL
LIN {X 0,Y 276.828,Z 773.78,A -85,B 0,C 180,E1 -17708.105,E2 -17708.105} C_VEL
LIN {X 0,Y 275.466,Z 785.369,A -85,B 0,C 180,E1 -17709.267,E2 -17709.267} C_VEL
LIN {X 0,Y 274.005,Z 796.686,A -85,B 0,C 180,E1 -17710.716,E2 -17710.716} C_VEL
LIN {X 0,Y 272.623,Z 806.871,A -85,B 0,C 180,E1 -17712.356,E2 -17712.356} C_VEL
LIN {X 0,Y 271.383,Z 816.183,A -85,B 0,C 180,E1 -17714.22,E2 -17714.22} C_VEL
LIN {X 0,Y 270.128,Z 825.195,A -85,B 0,C 180,E1 -17716.457,E2 -17716.457} C_VEL
LIN {X 0,Y 269.2,Z 832.358,A -85,B 0,C 180,E1 -17718.707,E2 -17718.707} C_VEL
LIN {X 0,Y 268.715,Z 838.065,A -85,B 0,C 180,E1 -17720.97,E2 -17720.97} C_VEL
LIN {X 0,Y 268.466,Z 842.498,A -85,B 0,C 180,E1 -17723.233,E2 -17723.233} C_VEL
LIN {X 0,Y 268.406,Z 845.782,A -85,B 0,C 180,E1 -17725.493,E2 -17725.493} C_VEL
LIN {X 0,Y 268.392,Z 847.38,A -85,B 0,C 180,E1 -17726.996,E2 -17726.996} C_VEL
LIN {X 0,Y 268.422,Z 848.539,A -85,B 0,C 180,E1 -17728.498,E2 -17728.498} C_VEL
LIN {X 0,Y 268.52,Z 849.226,A -85,B 0,C 180,E1 -17729.998,E2 -17729.998} C_VEL
LIN {X 0,Y 268.378,Z 849.478,A -85,B 0,C 180,E1 -17731.499,E2 -17731.499} C_VEL
LIN {X 0,Y 268.341,Z 849.328,A -85,B 0,C 180,E1 -17733.001,E2 -17733.001} C_VEL
LIN {X 0,Y 268.258,Z 848.199,A -85,B 0,C 180,E1 -17735.404,E2 -17735.404} C_VEL
LIN {X 0,Y 268.416,Z 846.317,A -85,B 0,C 180,E1 -17737.521,E2 -17737.521} C_VEL
LIN {X 0,Y 268.84,Z 843.37,A -85,B 0,C 180,E1 -17739.782,E2 -17739.782} C_VEL
LIN {X 0,Y 269.546,Z 839.384,A -85,B 0,C 180,E1 -17742.038,E2 -17742.038} C_VEL
LIN {X 0,Y 270.804,Z 834.296,A -85,B 0,C 180,E1 -17744.272,E2 -17744.272} C_VEL
LIN {X 0,Y 272.322,Z 827.947,A -85,B 0,C 180,E1 -17746.49,E2 -17746.49} C_VEL
LIN {X 0,Y 274.268,Z 820.121,A -85,B 0,C 180,E1 -17748.679,E2 -17748.679} C_VEL
LIN {X 0,Y 276.217,Z 812.177,A -85,B 0,C 180,E1 -17750.476,E2 -17750.476} C_VEL
LIN {X 0,Y 278.777,Z 801.472,A -85,B 0,C 180,E1 -17752.413,E2 -17752.413} C_VEL
LIN {X 0,Y 281.196,Z 790.748,A -85,B 0,C 180,E1 -17753.961,E2 -17753.961} C_VEL
LIN {X 0,Y 283.229,Z 780.521,A -85,B 0,C 180,E1 -17755.145,E2 -17755.145} C_VEL
LIN {X 0,Y 285.519,Z 767.45,A -85,B 0,C 180,E1 -17756.298,E2 -17756.298} C_VEL
LIN {X 0,Y 287.324,Z 754.321,A -85,B 0,C 180,E1 -17757.149,E2 -17757.149} C_VEL
LIN {X 0,Y 288.493,Z 741.161,A -85,B 0,C 180,E1 -17757.732,E2 -17757.732} C_VEL
LIN {X 0,Y 291.265,Z 688.813,A -85,B 0,C 180,E1 -17759.347,E2 -17759.347} C_VEL
LIN {X 0,Y 289.318,Z 670.091,A -85,B 0,C 180,E1 -17760.409,E2 -17760.409} C_VEL
LIN {X 0,Y 286.666,Z 654.615,A -85,B 0,C 180,E1 -17761.498,E2 -17761.498} C_VEL
LIN {X 0,Y 282.67,Z 645.825,A -85,B 0,C 180,E1 -17762.602,E2 -17762.602} C_VEL
LIN {X 0,Y 278.192,Z 636.969,A -85,B 0,C 180,E1 -17763.884,E2 -17763.884} C_VEL
LIN {X 0,Y 275.927,Z 632.486,A -85,B 0,C 180,E1 -17764.6,E2 -17764.6} C_VEL
LIN {X 0,Y 274.41,Z 626.145,A -85,B 0,C 180,E1 -17767.443,E2 -17767.443} C_VEL
LIN {X 0,Y 272.745,Z 619.987,A -85,B 0,C 180,E1 -17770.519,E2 -17770.519} C_VEL
LIN {X 0,Y 271.13,Z 614.83,A -85,B 0,C 180,E1 -17773.465,E2 -17773.465} C_VEL
LIN {X 0,Y 270.207,Z 611.83,A -85,B 0,C 180,E1 -17775.391,E2 -17775.391} C_VEL
LIN {X 0,Y 270.241,Z 611.822,A -85,B 0,C 180,E1 -17779.446,E2 -17779.446} C_VEL
LIN {X 0,Y 270.252,Z 611.816,A -85,B 0,C 180,E1 -17783.72,E2 -17783.72} C_VEL
LIN {X 0,Y 270.199,Z 611.825,A -85,B 0,C 180,E1 -17786.892,E2 -17786.892} C_VEL
LIN {X 0,Y 270.19,Z 611.824,A -85,B 0,C 180,E1 -17790.382,E2 -17790.382} C_VEL
LIN {X 0,Y 270.257,Z 611.812,A -85,B 0,C 180,E1 -17793.763,E2 -17793.763} C_VEL
LIN {X 0,Y 270.229,Z 611.817,A -85,B 0,C 180,E1 -17797.038,E2 -17797.038} C_VEL
LIN {X 0,Y 270.295,Z 611.811,A -85,B 0,C 180,E1 -17800.244,E2 -17800.244} C_VEL
LIN {X 0,Y 270.395,Z 611.798,A -85,B 0,C 180,E1 -17804.935,E2 -17804.935} C_VEL
LIN {X 0,Y 270.434,Z 611.798,A -85,B 0,C 180,E1 -17809.518,E2 -17809.518} C_VEL
LIN {X 0,Y 270.603,Z 611.774,A -85,B 0,C 180,E1 -17812.538,E2 -17812.538} C_VEL
LIN {X 0,Y 270.741,Z 611.881,A -85,B 0,C 180,E1 -17818.047,E2 -17818.047} C_VEL
LIN {X 0,Y 271.564,Z 614.16,A -85,B 0,C 180,E1 -17819.536,E2 -17819.536} C_VEL
LIN {X 0,Y 273.929,Z 617.85,A -85,B 0,C 180,E1 -17820.284,E2 -17820.284} C_VEL
LIN {X 0,Y 275.253,Z 619.862,A -85,B 0,C 180,E1 -17820.685,E2 -17820.685} C_VEL
LIN {X 0,Y 278.144,Z 624.496,A -85,B 0,C 180,E1 -17821.542,E2 -17821.542} C_VEL
LIN {X 0,Y 286.018,Z 637.612,A -85,B 0,C 180,E1 -17823.683,E2 -17823.683} C_VEL
LIN {X 0,Y 291.331,Z 648.784,A -85,B 0,C 180,E1 -17825.068,E2 -17825.068} C_VEL
LIN {X 0,Y 293.024,Z 652.683,A -85,B 0,C 180,E1 -17825.505,E2 -17825.505} C_VEL
LIN {X 0,Y 289.304,Z 718.159,A -85,B 0,C 180,E1 -17827.546,E2 -17827.546} C_VEL
LIN {X 0,Y 288.091,Z 731.742,A -85,B 0,C 180,E1 -17828.24,E2 -17828.24} C_VEL
LIN {X 0,Y 286.676,Z 744.182,A -85,B 0,C 180,E1 -17829.169,E2 -17829.169} C_VEL
LIN {X 0,Y 284.984,Z 755.054,A -85,B 0,C 180,E1 -17830.231,E2 -17830.231} C_VEL
LIN {X 0,Y 282.858,Z 766.407,A -85,B 0,C 180,E1 -17831.647,E2 -17831.647} C_VEL
LIN {X 0,Y 280.521,Z 777.427,A -85,B 0,C 180,E1 -17833.4,E2 -17833.4} C_VEL
LIN {X 0,Y 278.142,Z 786.848,A -85,B 0,C 180,E1 -17835.283,E2 -17835.283} C_VEL
LIN {X 0,Y 275.871,Z 795.379,A -85,B 0,C 180,E1 -17837.418,E2 -17837.418} C_VEL
LIN {X 0,Y 273.653,Z 803.039,A -85,B 0,C 180,E1 -17839.894,E2 -17839.894} C_VEL
LIN {X 0,Y 272.068,Z 808.526,A -85,B 0,C 180,E1 -17842.2,E2 -17842.2} C_VEL
LIN {X 0,Y 270.721,Z 813.005,A -85,B 0,C 180,E1 -17844.691,E2 -17844.691} C_VEL
LIN {X 0,Y 270.078,Z 815.101,A -85,B 0,C 180,E1 -17846.255,E2 -17846.255} C_VEL
LIN {X 0,Y 269.391,Z 816.905,A -85,B 0,C 180,E1 -17848.008,E2 -17848.008} C_VEL
LIN {X 0,Y 268.759,Z 818.398,A -85,B 0,C 180,E1 -17850.355,E2 -17850.355} C_VEL
LIN {X 0,Y 268.35,Z 818.876,A -85,B 0,C 180,E1 -17853.067,E2 -17853.067} C_VEL
LIN {X 0,Y 268.232,Z 818.034,A -85,B 0,C 180,E1 -17855.688,E2 -17855.688} C_VEL
LIN {X 0,Y 268.312,Z 816.044,A -85,B 0,C 180,E1 -17858.208,E2 -17858.208} C_VEL
LIN {X 0,Y 268.743,Z 812.681,A -85,B 0,C 180,E1 -17860.827,E2 -17860.827} C_VEL
LIN {X 0,Y 269.16,Z 808.753,A -85,B 0,C 180,E1 -17863.024,E2 -17863.024} C_VEL
LIN {X 0,Y 269.854,Z 803.438,A -85,B 0,C 180,E1 -17865.32,E2 -17865.32} C_VEL
LIN {X 0,Y 270.743,Z 796.89,A -85,B 0,C 180,E1 -17867.555,E2 -17867.555} C_VEL
LIN {X 0,Y 271.899,Z 788.81,A -85,B 0,C 180,E1 -17869.747,E2 -17869.747} C_VEL
LIN {X 0,Y 273.337,Z 778.92,A -85,B 0,C 180,E1 -17871.899,E2 -17871.899} C_VEL
LIN {X 0,Y 274.74,Z 768.563,A -85,B 0,C 180,E1 -17873.686,E2 -17873.686} C_VEL
LIN {X 0,Y 276.228,Z 756.844,A -85,B 0,C 180,E1 -17875.297,E2 -17875.297} C_VEL
LIN {X 0,Y 277.374,Z 745.831,A -85,B 0,C 180,E1 -17876.492,E2 -17876.492} C_VEL
LIN {X 0,Y 278.477,Z 732.719,A -85,B 0,C 180,E1 -17877.571,E2 -17877.571} C_VEL
LIN {X 0,Y 279.275,Z 719.587,A -85,B 0,C 180,E1 -17878.344,E2 -17878.344} C_VEL
LIN {X 0,Y 279.886,Z 704.088,A -85,B 0,C 180,E1 -17878.897,E2 -17878.897} C_VEL
LIN {X 0,Y 282.019,Z 642.555,A -85,B 0,C 180,E1 -17880.716,E2 -17880.716} C_VEL
LIN {X 0,Y 276.095,Z 626.421,A -85,B 0,C 180,E1 -17881.701,E2 -17881.701} C_VEL
LIN {X 0,Y 270.392,Z 612.32,A -85,B 0,C 180,E1 -17882.632,E2 -17882.632} C_VEL
LIN {X 0,Y 270.304,Z 611.814,A -85,B 0,C 180,E1 -17882.727,E2 -17882.727} C_VEL
LIN {X 0,Y 270.235,Z 611.822,A -85,B 0,C 180,E1 -17887.041,E2 -17887.041} C_VEL
LIN {X 0,Y 270.301,Z 611.816,A -85,B 0,C 180,E1 -17890.246,E2 -17890.246} C_VEL
LIN {X 0,Y 270.402,Z 611.8,A -85,B 0,C 180,E1 -17894.937,E2 -17894.937} C_VEL
LIN {X 0,Y 270.442,Z 611.795,A -85,B 0,C 180,E1 -17899.521,E2 -17899.521} C_VEL
LIN {X 0,Y 270.611,Z 611.779,A -85,B 0,C 180,E1 -17902.541,E2 -17902.541} C_VEL
LIN {X 0,Y 270.788,Z 611.756,A -85,B 0,C 180,E1 -17908.514,E2 -17908.514} C_VEL
LIN {X 0,Y 270.791,Z 611.751,A -85,B 0,C 180,E1 -17911.489,E2 -17911.489} C_VEL
LIN {X 0,Y 270.613,Z 611.773,A -85,B 0,C 180,E1 -17917.463,E2 -17917.463} C_VEL
LIN {X 0,Y 270.444,Z 611.797,A -85,B 0,C 180,E1 -17920.483,E2 -17920.483} C_VEL
LIN {X 0,Y 270.406,Z 611.802,A -85,B 0,C 180,E1 -17925.066,E2 -17925.066} C_VEL
LIN {X 0,Y 270.305,Z 611.806,A -85,B 0,C 180,E1 -17929.757,E2 -17929.757} C_VEL
LIN {X 0,Y 270.277,Z 611.817,A -85,B 0,C 180,E1 -17934.587,E2 -17934.587} C_VEL
LIN {X 0,Y 270.275,Z 611.815,A -85,B 0,C 180,E1 -17937.91,E2 -17937.91} C_VEL
LIN {X 0,Y 270.188,Z 611.824,A -85,B 0,C 180,E1 -17941.349,E2 -17941.349} C_VEL
LIN {X 0,Y 270.205,Z 611.817,A -85,B 0,C 180,E1 -17944.907,E2 -17944.907} C_VEL
LIN {X 0,Y 270.201,Z 611.823,A -85,B 0,C 180,E1 -17948.712,E2 -17948.712} C_VEL
LIN {X 0,Y 270.176,Z 611.832,A -85,B 0,C 180,E1 -17953.252,E2 -17953.252} C_VEL
LIN {X 0,Y 270.179,Z 611.827,A -85,B 0,C 180,E1 -17957.443,E2 -17957.443} C_VEL
LIN {X 0,Y 270.212,Z 611.817,A -85,B 0,C 180,E1 -17961.375,E2 -17961.375} C_VEL
LIN {X 0,Y 270.207,Z 611.817,A -85,B 0,C 180,E1 -17965.095,E2 -17965.095} C_VEL
LIN {X 0,Y 270.206,Z 611.823,A -85,B 0,C 180,E1 -17969.131,E2 -17969.131} C_VEL
LIN {X 0,Y 270.27,Z 611.818,A -85,B 0,C 180,E1 -17972.146,E2 -17972.146} C_VEL
LIN {X 0,Y 270.244,Z 611.822,A -85,B 0,C 180,E1 -17975.538,E2 -17975.538} C_VEL
LIN {X 0,Y 270.306,Z 611.806,A -85,B 0,C 180,E1 -17980.245,E2 -17980.245} C_VEL
LIN {X 0,Y 270.402,Z 611.79,A -85,B 0,C 180,E1 -17984.936,E2 -17984.936} C_VEL
LIN {X 0,Y 270.419,Z 611.796,A -85,B 0,C 180,E1 -17989.518,E2 -17989.518} C_VEL
LIN {X 0,Y 270.581,Z 611.777,A -85,B 0,C 180,E1 -17992.797,E2 -17992.797} C_VEL
LIN {X 0,Y 269.867,Z 611.871,A -85,B 0,C 180,E1 -17994.039,E2 -17994.039} C_VEL
LIN {X 0,Y 267.075,Z 612.218,A -85,B 0,C 180,E1 -17996.067,E2 -17996.067} C_VEL
LIN {X 0,Y 264.772,Z 612.5,A -85,B 0,C 180,E1 -17997.715,E2 -17997.715} C_VEL
LIN {X 0,Y 263.825,Z 612.614,A -85,B 0,C 180,E1 -17998.99,E2 -17998.99} C_VEL
LIN {X 0,Y 263.767,Z 612.621,A -85,B 0,C 180,E1 -17999.421,E2 -17999.421} C_VEL
LIN {X 0,Y 263.757,Z 612.619,A -85,B 0,C 180,E1 -18001.527,E2 -18001.527} C_VEL
LIN {X 0,Y 263.565,Z 612.651,A -85,B 0,C 180,E1 -18007.662,E2 -18007.662} C_VEL
LIN {X 0,Y 263.361,Z 612.678,A -85,B 0,C 180,E1 -18010.766,E2 -18010.766} C_VEL
LIN {X 0,Y 263.316,Z 612.677,A -85,B 0,C 180,E1 -18015.48,E2 -18015.48} C_VEL
LIN {X 0,Y 263.242,Z 612.695,A -85,B 0,C 180,E1 -18020.309,E2 -18020.309} C_VEL
LIN {X 0,Y 263.2,Z 612.695,A -85,B 0,C 180,E1 -18025.292,E2 -18025.292} C_VEL
LIN {X 0,Y 263.187,Z 612.704,A -85,B 0,C 180,E1 -18028.729,E2 -18028.729} C_VEL
LIN {X 0,Y 263.139,Z 612.706,A -85,B 0,C 180,E1 -18032.288,E2 -18032.288} C_VEL
LIN {X 0,Y 263.188,Z 612.703,A -85,B 0,C 180,E1 -18036.762,E2 -18036.762} C_VEL
LIN {X 0,Y 263.131,Z 612.708,A -85,B 0,C 180,E1 -18041.593,E2 -18041.593} C_VEL
LIN {X 0,Y 263.134,Z 612.706,A -85,B 0,C 180,E1 -18046.016,E2 -18046.016} C_VEL
LIN {X 0,Y 263.111,Z 612.709,A -85,B 0,C 180,E1 -18050.127,E2 -18050.127} C_VEL
LIN {X 0,Y 263.206,Z 612.762,A -85,B 0,C 180,E1 -18053.73,E2 -18053.73} C_VEL
LIN {X 0,Y 265.908,Z 625.455,A -85,B 0,C 180,E1 -18058.087,E2 -18058.087} C_VEL
LIN {X 0,Y 268.236,Z 637.048,A -85,B 0,C 180,E1 -18061.859,E2 -18061.859} C_VEL
LIN {X 0,Y 268.362,Z 637.968,A -85,B 0,C 180,E1 -18062.023,E2 -18062.023} C_VEL
LIN {X 0,Y 274.371,Z 688.275,A -85,B 0,C 180,E1 -18064.184,E2 -18064.184} C_VEL
LIN {X 0,Y 272.284,Z 746.691,A -85,B 0,C 180,E1 -18066.011,E2 -18066.011} C_VEL
LIN {X 0,Y 271.343,Z 760.45,A -85,B 0,C 180,E1 -18066.733,E2 -18066.733} C_VEL
LIN {X 0,Y 270.067,Z 772.425,A -85,B 0,C 180,E1 -18067.628,E2 -18067.628} C_VEL
LIN {X 0,Y 268.577,Z 784.998,A -85,B 0,C 180,E1 -18068.91,E2 -18068.91} C_VEL
LIN {X 0,Y 267.084,Z 796.304,A -85,B 0,C 180,E1 -18070.395,E2 -18070.395} C_VEL
LIN {X 0,Y 265.558,Z 807.185,A -85,B 0,C 180,E1 -18072.211,E2 -18072.211} C_VEL
LIN {X 0,Y 264.246,Z 816.617,A -85,B 0,C 180,E1 -18074.179,E2 -18074.179} C_VEL
LIN {X 0,Y 263.177,Z 824.1,A -85,B 0,C 180,E1 -18076.092,E2 -18076.092} C_VEL
LIN {X 0,Y 262.172,Z 831.427,A -85,B 0,C 180,E1 -18078.4,E2 -18078.4} C_VEL
LIN {X 0,Y 261.68,Z 837.242,A -85,B 0,C 180,E1 -18080.725,E2 -18080.725} C_VEL
LIN {X 0,Y 261.402,Z 841.767,A -85,B 0,C 180,E1 -18083.049,E2 -18083.049} C_VEL
LIN {X 0,Y 261.333,Z 845.136,A -85,B 0,C 180,E1 -18085.371,E2 -18085.371} C_VEL
LIN {X 0,Y 261.322,Z 846.775,A -85,B 0,C 180,E1 -18086.915,E2 -18086.915} C_VEL
LIN {X 0,Y 261.339,Z 847.982,A -85,B 0,C 180,E1 -18088.457,E2 -18088.457} C_VEL
LIN {X 0,Y 261.433,Z 848.742,A -85,B 0,C 180,E1 -18089.998,E2 -18089.998} C_VEL
LIN {X 0,Y 261.297,Z 849.033,A -85,B 0,C 180,E1 -18091.54,E2 -18091.54} C_VEL
LIN {X 0,Y 261.265,Z 848.92,A -85,B 0,C 180,E1 -18093.082,E2 -18093.082} C_VEL
LIN {X 0,Y 261.174,Z 847.99,A -85,B 0,C 180,E1 -18095.348,E2 -18095.348} C_VEL
LIN {X 0,Y 261.346,Z 846.055,A -85,B 0,C 180,E1 -18097.726,E2 -18097.726} C_VEL
LIN {X 0,Y 261.797,Z 843.201,A -85,B 0,C 180,E1 -18100.047,E2 -18100.047} C_VEL
LIN {X 0,Y 262.565,Z 839.324,A -85,B 0,C 180,E1 -18102.363,E2 -18102.363} C_VEL
LIN {X 0,Y 263.911,Z 834.332,A -85,B 0,C 180,E1 -18104.653,E2 -18104.653} C_VEL
LIN {X 0,Y 265.496,Z 828.082,A -85,B 0,C 180,E1 -18106.927,E2 -18106.927} C_VEL
LIN {X 0,Y 267.551,Z 820.37,A -85,B 0,C 180,E1 -18109.166,E2 -18109.166} C_VEL
LIN {X 0,Y 269.596,Z 812.616,A -85,B 0,C 180,E1 -18111.003,E2 -18111.003} C_VEL
LIN {X 0,Y 272.05,Z 803.294,A -85,B 0,C 180,E1 -18112.797,E2 -18112.797} C_VEL
LIN {X 0,Y 274.476,Z 793.042,A -85,B 0,C 180,E1 -18114.384,E2 -18114.384} C_VEL
LIN {X 0,Y 276.887,Z 781.833,A -85,B 0,C 180,E1 -18115.762,E2 -18115.762} C_VEL
LIN {X 0,Y 279.284,Z 769.427,A -85,B 0,C 180,E1 -18116.932,E2 -18116.932} C_VEL
LIN {X 0,Y 281.123,Z 757.072,A -85,B 0,C 180,E1 -18117.799,E2 -18117.799} C_VEL
LIN {X 0,Y 282.604,Z 742.803,A -85,B 0,C 180,E1 -18118.51,E2 -18118.51} C_VEL
LIN {X 0,Y 285.689,Z 689.843,A -85,B 0,C 180,E1 -18120.195,E2 -18120.195} C_VEL
LIN {X 0,Y 283.844,Z 671.563,A -85,B 0,C 180,E1 -18121.271,E2 -18121.271} C_VEL
LIN {X 0,Y 281.596,Z 657.92,A -85,B 0,C 180,E1 -18122.269,E2 -18122.269} C_VEL
LIN {X 0,Y 276.947,Z 647.509,A -85,B 0,C 180,E1 -18123.646,E2 -18123.646} C_VEL
LIN {X 0,Y 271.42,Z 636.922,A -85,B 0,C 180,E1 -18125.356,E2 -18125.356} C_VEL
LIN {X 0,Y 268.827,Z 632.156,A -85,B 0,C 180,E1 -18126.212,E2 -18126.212} C_VEL
LIN {X 0,Y 268.467,Z 630.908,A -85,B 0,C 180,E1 -18126.687,E2 -18126.687} C_VEL
LIN {X 0,Y 266.671,Z 624.006,A -85,B 0,C 180,E1 -18130.156,E2 -18130.156} C_VEL
LIN {X 0,Y 264.848,Z 618.059,A -85,B 0,C 180,E1 -18133.622,E2 -18133.622} C_VEL
LIN {X 0,Y 263.185,Z 612.703,A -85,B 0,C 180,E1 -18137.343,E2 -18137.343} C_VEL
LIN {X 0,Y 263.183,Z 612.703,A -85,B 0,C 180,E1 -18142.107,E2 -18142.107} C_VEL
LIN {X 0,Y 263.178,Z 612.696,A -85,B 0,C 180,E1 -18145.889,E2 -18145.889} C_VEL
LIN {X 0,Y 263.135,Z 612.703,A -85,B 0,C 180,E1 -18149.505,E2 -18149.505} C_VEL
LIN {X 0,Y 263.186,Z 612.697,A -85,B 0,C 180,E1 -18153.002,E2 -18153.002} C_VEL
LIN {X 0,Y 263.178,Z 612.696,A -85,B 0,C 180,E1 -18156.386,E2 -18156.386} C_VEL
LIN {X 0,Y 263.257,Z 612.686,A -85,B 0,C 180,E1 -18159.693,E2 -18159.693} C_VEL
LIN {X 0,Y 263.343,Z 612.678,A -85,B 0,C 180,E1 -18164.521,E2 -18164.521} C_VEL
LIN {X 0,Y 263.367,Z 612.68,A -85,B 0,C 180,E1 -18169.234,E2 -18169.234} C_VEL
LIN {X 0,Y 263.565,Z 612.651,A -85,B 0,C 180,E1 -18172.338,E2 -18172.338} C_VEL
LIN {X 0,Y 263.454,Z 612.772,A -85,B 0,C 180,E1 -18176.08,E2 -18176.08} C_VEL
LIN {X 0,Y 264.348,Z 614.92,A -85,B 0,C 180,E1 -18177.714,E2 -18177.714} C_VEL
LIN {X 0,Y 267.126,Z 618.88,A -85,B 0,C 180,E1 -18178.679,E2 -18178.679} C_VEL
LIN {X 0,Y 268.278,Z 620.343,A -85,B 0,C 180,E1 -18179.058,E2 -18179.058} C_VEL
LIN {X 0,Y 271.823,Z 625.779,A -85,B 0,C 180,E1 -18180.199,E2 -18180.199} C_VEL
LIN {X 0,Y 275.425,Z 631.61,A -85,B 0,C 180,E1 -18181.302,E2 -18181.302} C_VEL
LIN {X 0,Y 281.95,Z 642.981,A -85,B 0,C 180,E1 -18183.153,E2 -18183.153} C_VEL
LIN {X 0,Y 286.488,Z 652.784,A -85,B 0,C 180,E1 -18184.415,E2 -18184.415} C_VEL
LIN {X 0,Y 287.447,Z 655.216,A -85,B 0,C 180,E1 -18184.681,E2 -18184.681} C_VEL
LIN {X 0,Y 283.647,Z 718.441,A -85,B 0,C 180,E1 -18186.695,E2 -18186.695} C_VEL
LIN {X 0,Y 282.314,Z 732.35,A -85,B 0,C 180,E1 -18187.42,E2 -18187.42} C_VEL
LIN {X 0,Y 280.825,Z 744.665,A -85,B 0,C 180,E1 -18188.364,E2 -18188.364} C_VEL
LIN {X 0,Y 278.734,Z 757.244,A -85,B 0,C 180,E1 -18189.643,E2 -18189.643} C_VEL
LIN {X 0,Y 276.426,Z 768.904,A -85,B 0,C 180,E1 -18191.178,E2 -18191.178} C_VEL
LIN {X 0,Y 273.805,Z 779.972,A -85,B 0,C 180,E1 -18193.053,E2 -18193.053} C_VEL
LIN {X 0,Y 271.356,Z 789.156,A -85,B 0,C 180,E1 -18195.01,E2 -18195.01} C_VEL
LIN {X 0,Y 269.096,Z 796.89,A -85,B 0,C 180,E1 -18197.086,E2 -18197.086} C_VEL
LIN {X 0,Y 266.977,Z 803.706,A -85,B 0,C 180,E1 -18199.391,E2 -18199.391} C_VEL
LIN {X 0,Y 265.162,Z 809.531,A -85,B 0,C 180,E1 -18201.933,E2 -18201.933} C_VEL
LIN {X 0,Y 263.899,Z 813.469,A -85,B 0,C 180,E1 -18204.225,E2 -18204.225} C_VEL
LIN {X 0,Y 262.646,Z 816.854,A -85,B 0,C 180,E1 -18207.058,E2 -18207.058} C_VEL
LIN {X 0,Y 262.089,Z 818.244,A -85,B 0,C 180,E1 -18208.86,E2 -18208.86} C_VEL
LIN {X 0,Y 261.609,Z 819.073,A -85,B 0,C 180,E1 -18210.725,E2 -18210.725} C_VEL
LIN {X 0,Y 261.228,Z 819.202,A -85,B 0,C 180,E1 -18213.49,E2 -18213.49} C_VEL
LIN {X 0,Y 261.139,Z 818.002,A -85,B 0,C 180,E1 -18216.305,E2 -18216.305} C_VEL
LIN {X 0,Y 261.294,Z 815.821,A -85,B 0,C 180,E1 -18218.742,E2 -18218.742} C_VEL
LIN {X 0,Y 261.73,Z 812.413,A -85,B 0,C 180,E1 -18221.251,E2 -18221.251} C_VEL
LIN {X 0,Y 262.399,Z 806.875,A -85,B 0,C 180,E1 -18224.137,E2 -18224.137} C_VEL
LIN {X 0,Y 263.26,Z 800.418,A -85,B 0,C 180,E1 -18226.674,E2 -18226.674} C_VEL
LIN {X 0,Y 264.196,Z 793.865,A -85,B 0,C 180,E1 -18228.718,E2 -18228.718} C_VEL
LIN {X 0,Y 265.478,Z 785.284,A -85,B 0,C 180,E1 -18230.882,E2 -18230.882} C_VEL
LIN {X 0,Y 267.024,Z 774.863,A -85,B 0,C 180,E1 -18232.992,E2 -18232.992} C_VEL
LIN {X 0,Y 268.358,Z 764.871,A -85,B 0,C 180,E1 -18234.606,E2 -18234.606} C_VEL
LIN {X 0,Y 269.76,Z 753.311,A -85,B 0,C 180,E1 -18236.101,E2 -18236.101} C_VEL
LIN {X 0,Y 271.068,Z 740.677,A -85,B 0,C 180,E1 -18237.367,E2 -18237.367} C_VEL
LIN {X 0,Y 272.08,Z 726.924,A -85,B 0,C 180,E1 -18238.375,E2 -18238.375} C_VEL
LIN {X 0,Y 272.796,Z 713.57,A -85,B 0,C 180,E1 -18239.031,E2 -18239.031} C_VEL
LIN {X 0,Y 275.206,Z 643.816,A -85,B 0,C 180,E1 -18241.185,E2 -18241.185} C_VEL
LIN {X 0,Y 269.518,Z 628.336,A -85,B 0,C 180,E1 -18242.151,E2 -18242.151} C_VEL
LIN {X 0,Y 263.373,Z 613.447,A -85,B 0,C 180,E1 -18243.185,E2 -18243.185} C_VEL
LIN {X 0,Y 263.235,Z 612.705,A -85,B 0,C 180,E1 -18243.224,E2 -18243.224} C_VEL
LIN {X 0,Y 263.184,Z 612.703,A -85,B 0,C 180,E1 -18246.389,E2 -18246.389} C_VEL
LIN {X 0,Y 263.267,Z 612.692,A -85,B 0,C 180,E1 -18249.696,E2 -18249.696} C_VEL
LIN {X 0,Y 263.35,Z 612.681,A -85,B 0,C 180,E1 -18254.524,E2 -18254.524} C_VEL
LIN {X 0,Y 263.374,Z 612.675,A -85,B 0,C 180,E1 -18259.236,E2 -18259.236} C_VEL
LIN {X 0,Y 263.573,Z 612.655,A -85,B 0,C 180,E1 -18262.34,E2 -18262.34} C_VEL
LIN {X 0,Y 263.752,Z 612.633,A -85,B 0,C 180,E1 -18268.475,E2 -18268.475} C_VEL
LIN {X 0,Y 263.756,Z 612.628,A -85,B 0,C 180,E1 -18271.529,E2 -18271.529} C_VEL
LIN {X 0,Y 263.575,Z 612.65,A -85,B 0,C 180,E1 -18277.663,E2 -18277.663} C_VEL
LIN {X 0,Y 263.376,Z 612.679,A -85,B 0,C 180,E1 -18280.767,E2 -18280.767} C_VEL
LIN {X 0,Y 263.354,Z 612.678,A -85,B 0,C 180,E1 -18285.479,E2 -18285.479} C_VEL
LIN {X 0,Y 263.267,Z 612.682,A -85,B 0,C 180,E1 -18290.308,E2 -18290.308} C_VEL
LIN {X 0,Y 263.211,Z 612.698,A -85,B 0,C 180,E1 -18295.293,E2 -18295.293} C_VEL
LIN {X 0,Y 263.182,Z 612.701,A -85,B 0,C 180,E1 -18298.731,E2 -18298.731} C_VEL
LIN {X 0,Y 263.136,Z 612.699,A -85,B 0,C 180,E1 -18302.289,E2 -18302.289} C_VEL
LIN {X 0,Y 263.186,Z 612.694,A -85,B 0,C 180,E1 -18306.764,E2 -18306.764} C_VEL
LIN {X 0,Y 263.129,Z 612.708,A -85,B 0,C 180,E1 -18311.595,E2 -18311.595} C_VEL
LIN {X 0,Y 263.132,Z 612.703,A -85,B 0,C 180,E1 -18316.018,E2 -18316.018} C_VEL
LIN {X 0,Y 263.11,Z 612.699,A -85,B 0,C 180,E1 -18320.129,E2 -18320.129} C_VEL
LIN {X 0,Y 263.168,Z 612.693,A -85,B 0,C 180,E1 -18324.019,E2 -18324.019} C_VEL
LIN {X 0,Y 263.138,Z 612.705,A -85,B 0,C 180,E1 -18327.713,E2 -18327.713} C_VEL
LIN {X 0,Y 263.207,Z 612.7,A -85,B 0,C 180,E1 -18331.784,E2 -18331.784} C_VEL
LIN {X 0,Y 263.207,Z 612.697,A -85,B 0,C 180,E1 -18335.213,E2 -18335.213} C_VEL
LIN {X 0,Y 263.268,Z 612.687,A -85,B 0,C 180,E1 -18339.694,E2 -18339.694} C_VEL
LIN {X 0,Y 263.351,Z 612.668,A -85,B 0,C 180,E1 -18344.522,E2 -18344.522} C_VEL
LIN {X 0,Y 263.361,Z 612.674,A -85,B 0,C 180,E1 -18349.234,E2 -18349.234} C_VEL
LIN {X 0,Y 263.531,Z 612.656,A -85,B 0,C 180,E1 -18352.778,E2 -18352.778} C_VEL
LIN {X 0,Y 263.757,Z 612.625,A -85,B 0,C 180,E1 -18358.473,E2 -18358.473} C_VEL
LIN {X 0,Y 263.767,Z 612.621,A -85,B 0,C 180,E1 -18359.421,E2 -18359.421} C_VEL
LIN {X 0,Y 263.092,Z 612.707,A -85,B 0,C 180,E1 -18360.693,E2 -18360.693} C_VEL
LIN {X 0,Y 260.046,Z 613.084,A -85,B 0,C 180,E1 -18362.759,E2 -18362.759} C_VEL
LIN {X 0,Y 257.501,Z 613.407,A -85,B 0,C 180,E1 -18364.442,E2 -18364.442} C_VEL
LIN {X 0,Y 256.503,Z 613.53,A -85,B 0,C 180,E1 -18365.752,E2 -18365.752} C_VEL
LIN {X 0,Y 256.474,Z 613.536,A -85,B 0,C 180,E1 -18366.196,E2 -18366.196} C_VEL
LIN {X 0,Y 256.434,Z 613.54,A -85,B 0,C 180,E1 -18369.465,E2 -18369.465} C_VEL
LIN {X 0,Y 256.239,Z 613.564,A -85,B 0,C 180,E1 -18374.291,E2 -18374.291} C_VEL
LIN {X 0,Y 256.175,Z 613.571,A -85,B 0,C 180,E1 -18377.565,E2 -18377.565} C_VEL
LIN {X 0,Y 256.148,Z 613.578,A -85,B 0,C 180,E1 -18381.11,E2 -18381.11} C_VEL
LIN {X 0,Y 256.178,Z 613.571,A -85,B 0,C 180,E1 -18385.13,E2 -18385.13} C_VEL
LIN {X 0,Y 256.121,Z 613.58,A -85,B 0,C 180,E1 -18389.599,E2 -18389.599} C_VEL
LIN {X 0,Y 256.074,Z 613.585,A -85,B 0,C 180,E1 -18393.292,E2 -18393.292} C_VEL
LIN {X 0,Y 256.12,Z 613.581,A -85,B 0,C 180,E1 -18397.27,E2 -18397.27} C_VEL
LIN {X 0,Y 256.061,Z 613.591,A -85,B 0,C 180,E1 -18401.203,E2 -18401.203} C_VEL
LIN {X 0,Y 256.068,Z 613.588,A -85,B 0,C 180,E1 -18405.528,E2 -18405.528} C_VEL
LIN {X 0,Y 256.061,Z 613.59,A -85,B 0,C 180,E1 -18408.796,E2 -18408.796} C_VEL
LIN {X 0,Y 256.176,Z 613.656,A -85,B 0,C 180,E1 -18413.303,E2 -18413.303} C_VEL
LIN {X 0,Y 258.629,Z 625.219,A -85,B 0,C 180,E1 -18417.395,E2 -18417.395} C_VEL
LIN {X 0,Y 261.072,Z 637.08,A -85,B 0,C 180,E1 -18421.381,E2 -18421.381} C_VEL
LIN {X 0,Y 262.218,Z 642.184,A -85,B 0,C 180,E1 -18421.671,E2 -18421.671} C_VEL
LIN {X 0,Y 267.64,Z 688.968,A -85,B 0,C 180,E1 -18423.733,E2 -18423.733} C_VEL
LIN {X 0,Y 265.509,Z 746.079,A -85,B 0,C 180,E1 -18425.568,E2 -18425.568} C_VEL
LIN {X 0,Y 264.548,Z 759.885,A -85,B 0,C 180,E1 -18426.307,E2 -18426.307} C_VEL
LIN {X 0,Y 263.125,Z 772.907,A -85,B 0,C 180,E1 -18427.316,E2 -18427.316} C_VEL
LIN {X 0,Y 261.704,Z 784.497,A -85,B 0,C 180,E1 -18428.536,E2 -18428.536} C_VEL
LIN {X 0,Y 260.173,Z 795.821,A -85,B 0,C 180,E1 -18430.058,E2 -18430.058} C_VEL
LIN {X 0,Y 258.663,Z 806.476,A -85,B 0,C 180,E1 -18431.873,E2 -18431.873} C_VEL
LIN {X 0,Y 257.375,Z 815.336,A -85,B 0,C 180,E1 -18433.745,E2 -18433.745} C_VEL
LIN {X 0,Y 256.065,Z 824.356,A -85,B 0,C 180,E1 -18436.103,E2 -18436.103} C_VEL
LIN {X 0,Y 255.07,Z 831.521,A -85,B 0,C 180,E1 -18438.475,E2 -18438.475} C_VEL
LIN {X 0,Y 254.516,Z 838.058,A -85,B 0,C 180,E1 -18441.263,E2 -18441.263} C_VEL
LIN {X 0,Y 254.317,Z 842.295,A -85,B 0,C 180,E1 -18443.652,E2 -18443.652} C_VEL
LIN {X 0,Y 254.262,Z 844.488,A -85,B 0,C 180,E1 -18445.242,E2 -18445.242} C_VEL
LIN {X 0,Y 254.253,Z 846.171,A -85,B 0,C 180,E1 -18446.829,E2 -18446.829} C_VEL
LIN {X 0,Y 254.259,Z 847.419,A -85,B 0,C 180,E1 -18448.414,E2 -18448.414} C_VEL
LIN {X 0,Y 254.347,Z 848.245,A -85,B 0,C 180,E1 -18449.998,E2 -18449.998} C_VEL
LIN {X 0,Y 254.218,Z 848.588,A -85,B 0,C 180,E1 -18451.582,E2 -18451.582} C_VEL
LIN {X 0,Y 254.19,Z 848.513,A -85,B 0,C 180,E1 -18453.168,E2 -18453.168} C_VEL
LIN {X 0,Y 254.148,Z 847.15,A -85,B 0,C 180,E1 -18456.349,E2 -18456.349} C_VEL
LIN {X 0,Y 254.297,Z 845.821,A -85,B 0,C 180,E1 -18457.941,E2 -18457.941} C_VEL
LIN {X 0,Y 254.768,Z 843.054,A -85,B 0,C 180,E1 -18460.328,E2 -18460.328} C_VEL
LIN {X 0,Y 255.599,Z 839.266,A -85,B 0,C 180,E1 -18462.705,E2 -18462.705} C_VEL
LIN {X 0,Y 257.023,Z 834.368,A -85,B 0,C 180,E1 -18465.054,E2 -18465.054} C_VEL
LIN {X 0,Y 259.017,Z 827.23,A -85,B 0,C 180,E1 -18467.728,E2 -18467.728} C_VEL
LIN {X 0,Y 261.249,Z 819.331,A -85,B 0,C 180,E1 -18470.057,E2 -18470.057} C_VEL
LIN {X 0,Y 263.541,Z 811.45,A -85,B 0,C 180,E1 -18471.92,E2 -18471.92} C_VEL
LIN {X 0,Y 266.325,Z 800.86,A -85,B 0,C 180,E1 -18473.935,E2 -18473.935} C_VEL
LIN {X 0,Y 269.273,Z 788.919,A -85,B 0,C 180,E1 -18475.714,E2 -18475.714} C_VEL
LIN {X 0,Y 271.959,Z 776.795,A -85,B 0,C 180,E1 -18477.093,E2 -18477.093} C_VEL
LIN {X 0,Y 274.268,Z 764.183,A -85,B 0,C 180,E1 -18478.192,E2 -18478.192} C_VEL
LIN {X 0,Y 276.159,Z 751.021,A -85,B 0,C 180,E1 -18479.009,E2 -18479.009} C_VEL
LIN {X 0,Y 277.375,Z 737.688,A -85,B 0,C 180,E1 -18479.579,E2 -18479.579} C_VEL
LIN {X 0,Y 280.178,Z 690.657,A -85,B 0,C 180,E1 -18481.091,E2 -18481.091} C_VEL
LIN {X 0,Y 278.41,Z 672.503,A -85,B 0,C 180,E1 -18482.215,E2 -18482.215} C_VEL
LIN {X 0,Y 276.572,Z 661.082,A -85,B 0,C 180,E1 -18483.097,E2 -18483.097} C_VEL
LIN {X 0,Y 272.248,Z 651.417,A -85,B 0,C 180,E1 -18484.449,E2 -18484.449} C_VEL
LIN {X 0,Y 269.198,Z 645.353,A -85,B 0,C 180,E1 -18485.44,E2 -18485.44} C_VEL
LIN {X 0,Y 266.573,Z 640.5,A -85,B 0,C 180,E1 -18486.316,E2 -18486.316} C_VEL
LIN {X 0,Y 264.362,Z 636.368,A -85,B 0,C 180,E1 -18487.103,E2 -18487.103} C_VEL
LIN {X 0,Y 261.469,Z 631.444,A -85,B 0,C 180,E1 -18488.159,E2 -18488.159} C_VEL
LIN {X 0,Y 261.215,Z 630.668,A -85,B 0,C 180,E1 -18488.397,E2 -18488.397} C_VEL
LIN {X 0,Y 259.53,Z 624.402,A -85,B 0,C 180,E1 -18491.868,E2 -18491.868} C_VEL
LIN {X 0,Y 257.707,Z 618.614,A -85,B 0,C 180,E1 -18495.646,E2 -18495.646} C_VEL
LIN {X 0,Y 256.105,Z 613.584,A -85,B 0,C 180,E1 -18499.669,E2 -18499.669} C_VEL
LIN {X 0,Y 256.15,Z 613.575,A -85,B 0,C 180,E1 -18502.87,E2 -18502.87} C_VEL
LIN {X 0,Y 256.079,Z 613.582,A -85,B 0,C 180,E1 -18506.709,E2 -18506.709} C_VEL
LIN {X 0,Y 256.121,Z 613.572,A -85,B 0,C 180,E1 -18511.408,E2 -18511.408} C_VEL
LIN {X 0,Y 256.161,Z 613.574,A -85,B 0,C 180,E1 -18515.698,E2 -18515.698} C_VEL
LIN {X 0,Y 256.162,Z 613.571,A -85,B 0,C 180,E1 -18519.104,E2 -18519.104} C_VEL
LIN {X 0,Y 256.292,Z 613.56,A -85,B 0,C 180,E1 -18524.084,E2 -18524.084} C_VEL
LIN {X 0,Y 256.303,Z 613.56,A -85,B 0,C 180,E1 -18528.933,E2 -18528.933} C_VEL
LIN {X 0,Y 256.532,Z 613.528,A -85,B 0,C 180,E1 -18532.127,E2 -18532.127} C_VEL
LIN {X 0,Y 256.504,Z 613.691,A -85,B 0,C 180,E1 -18533.905,E2 -18533.905} C_VEL
LIN {X 0,Y 257.002,Z 615.761,A -85,B 0,C 180,E1 -18535.589,E2 -18535.589} C_VEL
LIN {X 0,Y 259.971,Z 619.739,A -85,B 0,C 180,E1 -18536.755,E2 -18536.755} C_VEL
LIN {X 0,Y 261.56,Z 621.551,A -85,B 0,C 180,E1 -18537.328,E2 -18537.328} C_VEL
LIN {X 0,Y 265.121,Z 626.49,A -85,B 0,C 180,E1 -18538.578,E2 -18538.578} C_VEL
LIN {X 0,Y 269.384,Z 633.026,A -85,B 0,C 180,E1 -18540,E2 -18540} C_VEL
LIN {X 0,Y 277.368,Z 647.159,A -85,B 0,C 180,E1 -18542.445,E2 -18542.445} C_VEL
LIN {X 0,Y 281.899,Z 657.184,A -85,B 0,C 180,E1 -18543.78,E2 -18543.78} C_VEL
LIN {X 0,Y 278.023,Z 719.458,A -85,B 0,C 180,E1 -18545.833,E2 -18545.833} C_VEL
LIN {X 0,Y 276.634,Z 733.257,A -85,B 0,C 180,E1 -18546.573,E2 -18546.573} C_VEL
LIN {X 0,Y 275.073,Z 745.371,A -85,B 0,C 180,E1 -18547.524,E2 -18547.524} C_VEL
LIN {X 0,Y 273.054,Z 756.821,A -85,B 0,C 180,E1 -18548.697,E2 -18548.697} C_VEL
LIN {X 0,Y 270.515,Z 768.879,A -85,B 0,C 180,E1 -18550.293,E2 -18550.293} C_VEL
LIN {X 0,Y 267.921,Z 779.504,A -85,B 0,C 180,E1 -18552.114,E2 -18552.114} C_VEL
LIN {X 0,Y 265.638,Z 787.483,A -85,B 0,C 180,E1 -18553.775,E2 -18553.775} C_VEL
LIN {X 0,Y 263.134,Z 795.875,A -85,B 0,C 180,E1 -18555.954,E2 -18555.954} C_VEL
LIN {X 0,Y 261.078,Z 802.27,A -85,B 0,C 180,E1 -18558.033,E2 -18558.033} C_VEL
LIN {X 0,Y 258.923,Z 808.575,A -85,B 0,C 180,E1 -18560.662,E2 -18560.662} C_VEL
LIN {X 0,Y 257.256,Z 813.331,A -85,B 0,C 180,E1 -18563.336,E2 -18563.336} C_VEL
LIN {X 0,Y 255.975,Z 816.765,A -85,B 0,C 180,E1 -18566.059,E2 -18566.059} C_VEL
LIN {X 0,Y 255.19,Z 818.516,A -85,B 0,C 180,E1 -18568.206,E2 -18568.206} C_VEL
LIN {X 0,Y 254.463,Z 819.691,A -85,B 0,C 180,E1 -18571.113,E2 -18571.113} C_VEL
LIN {X 0,Y 254.097,Z 819.492,A -85,B 0,C 180,E1 -18573.929,E2 -18573.929} C_VEL
LIN {X 0,Y 254.042,Z 818.054,A -85,B 0,C 180,E1 -18576.655,E2 -18576.655} C_VEL
LIN {X 0,Y 254.292,Z 815.271,A -85,B 0,C 180,E1 -18579.469,E2 -18579.469} C_VEL
LIN {X 0,Y 254.732,Z 811.807,A -85,B 0,C 180,E1 -18581.85,E2 -18581.85} C_VEL
LIN {X 0,Y 255.358,Z 807.034,A -85,B 0,C 180,E1 -18584.312,E2 -18584.312} C_VEL
LIN {X 0,Y 256.154,Z 801.118,A -85,B 0,C 180,E1 -18586.695,E2 -18586.695} C_VEL
LIN {X 0,Y 257.231,Z 793.804,A -85,B 0,C 180,E1 -18589.028,E2 -18589.028} C_VEL
LIN {X 0,Y 258.633,Z 784.803,A -85,B 0,C 180,E1 -18591.321,E2 -18591.321} C_VEL
LIN {X 0,Y 260.052,Z 775.433,A -85,B 0,C 180,E1 -18593.249,E2 -18593.249} C_VEL
LIN {X 0,Y 261.538,Z 764.524,A -85,B 0,C 180,E1 -18595.043,E2 -18595.043} C_VEL
LIN {X 0,Y 263.018,Z 752.452,A -85,B 0,C 180,E1 -18596.618,E2 -18596.618} C_VEL
LIN {X 0,Y 264.323,Z 739.76,A -85,B 0,C 180,E1 -18597.877,E2 -18597.877} C_VEL
LIN {X 0,Y 265.346,Z 726.07,A -85,B 0,C 180,E1 -18598.878,E2 -18598.878} C_VEL
LIN {X 0,Y 266.054,Z 712.577,A -85,B 0,C 180,E1 -18599.52,E2 -18599.52} C_VEL
LIN {X 0,Y 268.633,Z 645.579,A -85,B 0,C 180,E1 -18601.627,E2 -18601.627} C_VEL
LIN {X 0,Y 262.632,Z 629.645,A -85,B 0,C 180,E1 -18602.673,E2 -18602.673} C_VEL
LIN {X 0,Y 256.222,Z 613.782,A -85,B 0,C 180,E1 -18603.806,E2 -18603.806} C_VEL
LIN {X 0,Y 256.176,Z 613.576,A -85,B 0,C 180,E1 -18603.965,E2 -18603.965} C_VEL
LIN {X 0,Y 256.184,Z 613.573,A -85,B 0,C 180,E1 -18608.865,E2 -18608.865} C_VEL
LIN {X 0,Y 256.281,Z 613.56,A -85,B 0,C 180,E1 -18613.699,E2 -18613.699} C_VEL
LIN {X 0,Y 256.295,Z 613.557,A -85,B 0,C 180,E1 -18617.33,E2 -18617.33} C_VEL
LIN {X 0,Y 256.496,Z 613.536,A -85,B 0,C 180,E1 -18620.539,E2 -18620.539} C_VEL
LIN {X 0,Y 256.488,Z 613.535,A -85,B 0,C 180,E1 -18623.709,E2 -18623.709} C_VEL
LIN {X 0,Y 256.715,Z 613.509,A -85,B 0,C 180,E1 -18628.433,E2 -18628.433} C_VEL
LIN {X 0,Y 256.718,Z 613.505,A -85,B 0,C 180,E1 -18631.57,E2 -18631.57} C_VEL
LIN {X 0,Y 256.542,Z 613.526,A -85,B 0,C 180,E1 -18637.875,E2 -18637.875} C_VEL
LIN {X 0,Y 256.312,Z 613.556,A -85,B 0,C 180,E1 -18641.068,E2 -18641.068} C_VEL
LIN {X 0,Y 256.303,Z 613.555,A -85,B 0,C 180,E1 -18645.916,E2 -18645.916} C_VEL
LIN {X 0,Y 256.17,Z 613.57,A -85,B 0,C 180,E1 -18650.896,E2 -18650.896} C_VEL
LIN {X 0,Y 256.191,Z 613.574,A -85,B 0,C 180,E1 -18655.14,E2 -18655.14} C_VEL
LIN {X 0,Y 256.117,Z 613.577,A -85,B 0,C 180,E1 -18659.601,E2 -18659.601} C_VEL
LIN {X 0,Y 256.071,Z 613.576,A -85,B 0,C 180,E1 -18663.294,E2 -18663.294} C_VEL
LIN {X 0,Y 256.118,Z 613.578,A -85,B 0,C 180,E1 -18667.272,E2 -18667.272} C_VEL
LIN {X 0,Y 256.059,Z 613.589,A -85,B 0,C 180,E1 -18671.204,E2 -18671.204} C_VEL
LIN {X 0,Y 256.067,Z 613.586,A -85,B 0,C 180,E1 -18675.53,E2 -18675.53} C_VEL
LIN {X 0,Y 256.06,Z 613.581,A -85,B 0,C 180,E1 -18678.798,E2 -18678.798} C_VEL
LIN {X 0,Y 256.135,Z 613.561,A -85,B 0,C 180,E1 -18682.868,E2 -18682.868} C_VEL
LIN {X 0,Y 256.082,Z 613.578,A -85,B 0,C 180,E1 -18686.709,E2 -18686.709} C_VEL
LIN {X 0,Y 256.144,Z 613.578,A -85,B 0,C 180,E1 -18691.405,E2 -18691.405} C_VEL
LIN {X 0,Y 256.148,Z 613.579,A -85,B 0,C 180,E1 -18695.697,E2 -18695.697} C_VEL
LIN {X 0,Y 256.168,Z 613.569,A -85,B 0,C 180,E1 -18699.105,E2 -18699.105} C_VEL
LIN {X 0,Y 256.286,Z 613.548,A -85,B 0,C 180,E1 -18704.084,E2 -18704.084} C_VEL
LIN {X 0,Y 256.3,Z 613.55,A -85,B 0,C 180,E1 -18707.328,E2 -18707.328} C_VEL
LIN {X 0,Y 256.522,Z 613.533,A -85,B 0,C 180,E1 -18712.127,E2 -18712.127} C_VEL
LIN {X 0,Y 256.504,Z 613.529,A -85,B 0,C 180,E1 -18716.859,E2 -18716.859} C_VEL
LIN {X 0,Y 256.771,Z 613.495,A -85,B 0,C 180,E1 -18720,E2 -18720} C_VEL
LIN {X 0,Y 256.504,Z 613.524,A -85,B 0,C 180,E1 -18723.142,E2 -18723.142} C_VEL
LIN {X 0,Y 256.474,Z 613.536,A -85,B 0,C 180,E1 -18726.196,E2 -18726.196} C_VEL
LIN {X 0,Y 255.931,Z 613.613,A -85,B 0,C 180,E1 -18727.505,E2 -18727.505} C_VEL
LIN {X 0,Y 254.365,Z 613.812,A -85,B 0,C 180,E1 -18728.789,E2 -18728.789} C_VEL
LIN {X 0,Y 250.485,Z 614.289,A -85,B 0,C 180,E1 -18731.369,E2 -18731.369} C_VEL
LIN {X 0,Y 249.327,Z 614.425,A -85,B 0,C 180,E1 -18732.717,E2 -18732.717} C_VEL
LIN {X 0,Y 249.208,Z 614.436,A -85,B 0,C 180,E1 -18733.176,E2 -18733.176} C_VEL
LIN {X 0,Y 249.179,Z 614.442,A -85,B 0,C 180,E1 -18736.468,E2 -18736.468} C_VEL
LIN {X 0,Y 249.087,Z 614.456,A -85,B 0,C 180,E1 -18741.518,E2 -18741.518} C_VEL
LIN {X 0,Y 249.124,Z 614.448,A -85,B 0,C 180,E1 -18745.475,E2 -18745.475} C_VEL
LIN {X 0,Y 249.091,Z 614.459,A -85,B 0,C 180,E1 -18748.993,E2 -18748.993} C_VEL
LIN {X 0,Y 249.037,Z 614.463,A -85,B 0,C 180,E1 -18752.425,E2 -18752.425} C_VEL
LIN {X 0,Y 249.054,Z 614.461,A -85,B 0,C 180,E1 -18756.342,E2 -18756.342} C_VEL
LIN {X 0,Y 249.012,Z 614.467,A -85,B 0,C 180,E1 -18760.477,E2 -18760.477} C_VEL
LIN {X 0,Y 249.014,Z 614.47,A -85,B 0,C 180,E1 -18764.877,E2 -18764.877} C_VEL
LIN {X 0,Y 249.024,Z 614.466,A -85,B 0,C 180,E1 -18767.362,E2 -18767.362} C_VEL
LIN {X 0,Y 249.049,Z 614.462,A -85,B 0,C 180,E1 -18772.199,E2 -18772.199} C_VEL
LIN {X 0,Y 249.106,Z 614.511,A -85,B 0,C 180,E1 -18772.846,E2 -18772.846} C_VEL
LIN {X 0,Y 251.512,Z 625.786,A -85,B 0,C 180,E1 -18776.961,E2 -18776.961} C_VEL
LIN {X 0,Y 253.771,Z 636.712,A -85,B 0,C 180,E1 -18780.747,E2 -18780.747} C_VEL
LIN {X 0,Y 255.619,Z 643.241,A -85,B 0,C 180,E1 -18781.151,E2 -18781.151} C_VEL
LIN {X 0,Y 260.938,Z 689.221,A -85,B 0,C 180,E1 -18783.244,E2 -18783.244} C_VEL
LIN {X 0,Y 258.667,Z 746.484,A -85,B 0,C 180,E1 -18785.146,E2 -18785.146} C_VEL
LIN {X 0,Y 257.69,Z 760.029,A -85,B 0,C 180,E1 -18785.904,E2 -18785.904} C_VEL
LIN {X 0,Y 256.301,Z 772.384,A -85,B 0,C 180,E1 -18786.891,E2 -18786.891} C_VEL
LIN {X 0,Y 254.843,Z 783.995,A -85,B 0,C 180,E1 -18788.141,E2 -18788.141} C_VEL
LIN {X 0,Y 253.271,Z 795.338,A -85,B 0,C 180,E1 -18789.703,E2 -18789.703} C_VEL
LIN {X 0,Y 251.79,Z 805.623,A -85,B 0,C 180,E1 -18791.487,E2 -18791.487} C_VEL
LIN {X 0,Y 250.479,Z 814.076,A -85,B 0,C 180,E1 -18793.291,E2 -18793.291} C_VEL
LIN {X 0,Y 249.111,Z 823.218,A -85,B 0,C 180,E1 -18795.707,E2 -18795.707} C_VEL
LIN {X 0,Y 248.055,Z 830.563,A -85,B 0,C 180,E1 -18798.145,E2 -18798.145} C_VEL
LIN {X 0,Y 247.582,Z 835.511,A -85,B 0,C 180,E1 -18800.192,E2 -18800.192} C_VEL
LIN {X 0,Y 247.27,Z 840.261,A -85,B 0,C 180,E1 -18802.65,E2 -18802.65} C_VEL
LIN {X 0,Y 247.196,Z 843.814,A -85,B 0,C 180,E1 -18805.105,E2 -18805.105} C_VEL
LIN {X 0,Y 247.186,Z 845.558,A -85,B 0,C 180,E1 -18806.738,E2 -18806.738} C_VEL
LIN {X 0,Y 247.182,Z 846.845,A -85,B 0,C 180,E1 -18808.369,E2 -18808.369} C_VEL
LIN {X 0,Y 247.264,Z 847.714,A -85,B 0,C 180,E1 -18809.998,E2 -18809.998} C_VEL
LIN {X 0,Y 247.141,Z 848.137,A -85,B 0,C 180,E1 -18811.628,E2 -18811.628} C_VEL
LIN {X 0,Y 247.093,Z 848.107,A -85,B 0,C 180,E1 -18813.259,E2 -18813.259} C_VEL
LIN {X 0,Y 247.06,Z 846.831,A -85,B 0,C 180,E1 -18816.532,E2 -18816.532} C_VEL
LIN {X 0,Y 247.224,Z 845.584,A -85,B 0,C 180,E1 -18818.17,E2 -18818.17} C_VEL
LIN {X 0,Y 247.759,Z 842.892,A -85,B 0,C 180,E1 -18820.623,E2 -18820.623} C_VEL
LIN {X 0,Y 248.642,Z 839.208,A -85,B 0,C 180,E1 -18823.067,E2 -18823.067} C_VEL
LIN {X 0,Y 250.154,Z 834.449,A -85,B 0,C 180,E1 -18825.478,E2 -18825.478} C_VEL
LIN {X 0,Y 251.931,Z 828.483,A -85,B 0,C 180,E1 -18827.868,E2 -18827.868} C_VEL
LIN {X 0,Y 254.188,Z 821.079,A -85,B 0,C 180,E1 -18830.217,E2 -18830.217} C_VEL
LIN {X 0,Y 256.987,Z 811.977,A -85,B 0,C 180,E1 -18832.509,E2 -18832.509} C_VEL
LIN {X 0,Y 259.906,Z 801.753,A -85,B 0,C 180,E1 -18834.564,E2 -18834.564} C_VEL
LIN {X 0,Y 262.97,Z 790.152,A -85,B 0,C 180,E1 -18836.377,E2 -18836.377} C_VEL
LIN {X 0,Y 265.731,Z 778.572,A -85,B 0,C 180,E1 -18837.782,E2 -18837.782} C_VEL
LIN {X 0,Y 268.333,Z 765.445,A -85,B 0,C 180,E1 -18838.98,E2 -18838.98} C_VEL
LIN {X 0,Y 270.429,Z 752.223,A -85,B 0,C 180,E1 -18839.855,E2 -18839.855} C_VEL
LIN {X 0,Y 271.735,Z 739.354,A -85,B 0,C 180,E1 -18840.446,E2 -18840.446} C_VEL
LIN {X 0,Y 274.798,Z 691.513,A -85,B 0,C 180,E1 -18842.042,E2 -18842.042} C_VEL
LIN {X 0,Y 273.24,Z 674.569,A -85,B 0,C 180,E1 -18843.129,E2 -18843.129} C_VEL
LIN {X 0,Y 271.633,Z 664.247,A -85,B 0,C 180,E1 -18843.95,E2 -18843.95} C_VEL
LIN {X 0,Y 266.179,Z 652.001,A -85,B 0,C 180,E1 -18845.806,E2 -18845.806} C_VEL
LIN {X 0,Y 260.773,Z 641.726,A -85,B 0,C 180,E1 -18847.757,E2 -18847.757} C_VEL
LIN {X 0,Y 257.145,Z 635.676,A -85,B 0,C 180,E1 -18849.147,E2 -18849.147} C_VEL
LIN {X 0,Y 254.357,Z 631.019,A -85,B 0,C 180,E1 -18850.309,E2 -18850.309} C_VEL
LIN {X 0,Y 253.945,Z 630.047,A -85,B 0,C 180,E1 -18850.538,E2 -18850.538} C_VEL
LIN {X 0,Y 251.992,Z 623.535,A -85,B 0,C 180,E1 -18854.694,E2 -18854.694} C_VEL
LIN {X 0,Y 250.739,Z 619.503,A -85,B 0,C 180,E1 -18857.724,E2 -18857.724} C_VEL
LIN {X 0,Y 249.997,Z 617.203,A -85,B 0,C 180,E1 -18859.715,E2 -18859.715} C_VEL
LIN {X 0,Y 249.076,Z 614.458,A -85,B 0,C 180,E1 -18862.551,E2 -18862.551} C_VEL
LIN {X 0,Y 249.056,Z 614.455,A -85,B 0,C 180,E1 -18865.641,E2 -18865.641} C_VEL
LIN {X 0,Y 249.042,Z 614.458,A -85,B 0,C 180,E1 -18869.471,E2 -18869.471} C_VEL
LIN {X 0,Y 249.066,Z 614.454,A -85,B 0,C 180,E1 -18873.161,E2 -18873.161} C_VEL
LIN {X 0,Y 249.074,Z 614.451,A -85,B 0,C 180,E1 -18876.732,E2 -18876.732} C_VEL
LIN {X 0,Y 249.104,Z 614.45,A -85,B 0,C 180,E1 -18880.211,E2 -18880.211} C_VEL
LIN {X 0,Y 249.235,Z 614.44,A -85,B 0,C 180,E1 -18883.621,E2 -18883.621} C_VEL
LIN {X 0,Y 249.246,Z 614.436,A -85,B 0,C 180,E1 -18888.616,E2 -18888.616} C_VEL
LIN {X 0,Y 249.461,Z 614.522,A -85,B 0,C 180,E1 -18891.105,E2 -18891.105} C_VEL
LIN {X 0,Y 250.142,Z 616.736,A -85,B 0,C 180,E1 -18893.268,E2 -18893.268} C_VEL
LIN {X 0,Y 252.989,Z 620.781,A -85,B 0,C 180,E1 -18894.59,E2 -18894.59} C_VEL
LIN {X 0,Y 254.698,Z 622.767,A -85,B 0,C 180,E1 -18895.301,E2 -18895.301} C_VEL
LIN {X 0,Y 257.826,Z 626.528,A -85,B 0,C 180,E1 -18896.532,E2 -18896.532} C_VEL
LIN {X 0,Y 261.838,Z 632.316,A -85,B 0,C 180,E1 -18898.029,E2 -18898.029} C_VEL
LIN {X 0,Y 265.651,Z 638.343,A -85,B 0,C 180,E1 -18899.375,E2 -18899.375} C_VEL
LIN {X 0,Y 273.204,Z 652.12,A -85,B 0,C 180,E1 -18901.827,E2 -18901.827} C_VEL
LIN {X 0,Y 276.558,Z 659.594,A -85,B 0,C 180,E1 -18902.863,E2 -18902.863} C_VEL
LIN {X 0,Y 272.566,Z 719.926,A -85,B 0,C 180,E1 -18904.899,E2 -18904.899} C_VEL
LIN {X 0,Y 271.138,Z 733.259,A -85,B 0,C 180,E1 -18905.624,E2 -18905.624} C_VEL
LIN {X 0,Y 269.474,Z 745.529,A -85,B 0,C 180,E1 -18906.598,E2 -18906.598} C_VEL
LIN {X 0,Y 267.413,Z 756.688,A -85,B 0,C 180,E1 -18907.741,E2 -18907.741} C_VEL
LIN {X 0,Y 265.074,Z 767.447,A -85,B 0,C 180,E1 -18909.153,E2 -18909.153} C_VEL
LIN {X 0,Y 262.351,Z 778.512,A -85,B 0,C 180,E1 -18911.003,E2 -18911.003} C_VEL
LIN {X 0,Y 259.566,Z 787.666,A -85,B 0,C 180,E1 -18912.916,E2 -18912.916} C_VEL
LIN {X 0,Y 256.971,Z 795.797,A -85,B 0,C 180,E1 -18915.059,E2 -18915.059} C_VEL
LIN {X 0,Y 254.695,Z 802.48,A -85,B 0,C 180,E1 -18917.255,E2 -18917.255} C_VEL
LIN {X 0,Y 252.729,Z 807.913,A -85,B 0,C 180,E1 -18919.493,E2 -18919.493} C_VEL
LIN {X 0,Y 250.764,Z 813.174,A -85,B 0,C 180,E1 -18922.357,E2 -18922.357} C_VEL
LIN {X 0,Y 249.135,Z 817.129,A -85,B 0,C 180,E1 -18925.489,E2 -18925.489} C_VEL
LIN {X 0,Y 248,Z 819.399,A -85,B 0,C 180,E1 -18928.543,E2 -18928.543} C_VEL
LIN {X 0,Y 247.32,Z 820.186,A -85,B 0,C 180,E1 -18931.519,E2 -18931.519} C_VEL
LIN {X 0,Y 246.976,Z 819.557,A -85,B 0,C 180,E1 -18934.689,E2 -18934.689} C_VEL
LIN {X 0,Y 246.965,Z 817.951,A -85,B 0,C 180,E1 -18937.177,E2 -18937.177} C_VEL
LIN {X 0,Y 247.27,Z 815.085,A -85,B 0,C 180,E1 -18939.882,E2 -18939.882} C_VEL
LIN {X 0,Y 247.856,Z 810.373,A -85,B 0,C 180,E1 -18942.884,E2 -18942.884} C_VEL
LIN {X 0,Y 248.626,Z 804.753,A -85,B 0,C 180,E1 -18945.541,E2 -18945.541} C_VEL
LIN {X 0,Y 249.508,Z 798.628,A -85,B 0,C 180,E1 -18947.823,E2 -18947.823} C_VEL
LIN {X 0,Y 250.711,Z 790.849,A -85,B 0,C 180,E1 -18950.152,E2 -18950.152} C_VEL
LIN {X 0,Y 252.217,Z 781.433,A -85,B 0,C 180,E1 -18952.408,E2 -18952.408} C_VEL
LIN {X 0,Y 253.785,Z 770.843,A -85,B 0,C 180,E1 -18954.443,E2 -18954.443} C_VEL
LIN {X 0,Y 255.441,Z 759.097,A -85,B 0,C 180,E1 -18956.213,E2 -18956.213} C_VEL
LIN {X 0,Y 256.749,Z 747.57,A -85,B 0,C 180,E1 -18957.59,E2 -18957.59} C_VEL
LIN {X 0,Y 257.988,Z 734.783,A -85,B 0,C 180,E1 -18958.74,E2 -18958.74} C_VEL
LIN {X 0,Y 258.859,Z 721.378,A -85,B 0,C 180,E1 -18959.613,E2 -18959.613} C_VEL
LIN {X 0,Y 259.534,Z 706.217,A -85,B 0,C 180,E1 -18960.217,E2 -18960.217} C_VEL
LIN {X 0,Y 261.783,Z 646.565,A -85,B 0,C 180,E1 -18962.143,E2 -18962.143} C_VEL
LIN {X 0,Y 255.606,Z 630.501,A -85,B 0,C 180,E1 -18963.243,E2 -18963.243} C_VEL
LIN {X 0,Y 249.189,Z 614.863,A -85,B 0,C 180,E1 -18964.4,E2 -18964.4} C_VEL
LIN {X 0,Y 249.154,Z 614.449,A -85,B 0,C 180,E1 -18964.481,E2 -18964.481} C_VEL
LIN {X 0,Y 249.125,Z 614.454,A -85,B 0,C 180,E1 -18968.584,E2 -18968.584} C_VEL
LIN {X 0,Y 249.24,Z 614.437,A -85,B 0,C 180,E1 -18973.624,E2 -18973.624} C_VEL
LIN {X 0,Y 249.253,Z 614.437,A -85,B 0,C 180,E1 -18978.618,E2 -18978.618} C_VEL
LIN {X 0,Y 249.484,Z 614.408,A -85,B 0,C 180,E1 -18981.905,E2 -18981.905} C_VEL
LIN {X 0,Y 249.439,Z 614.415,A -85,B 0,C 180,E1 -18986.771,E2 -18986.771} C_VEL
LIN {X 0,Y 249.729,Z 614.377,A -85,B 0,C 180,E1 -18990.002,E2 -18990.002} C_VEL
LIN {X 0,Y 249.443,Z 614.412,A -85,B 0,C 180,E1 -18993.232,E2 -18993.232} C_VEL
LIN {X 0,Y 249.486,Z 614.406,A -85,B 0,C 180,E1 -18998.099,E2 -18998.099} C_VEL
LIN {X 0,Y 249.255,Z 614.434,A -85,B 0,C 180,E1 -19001.385,E2 -19001.385} C_VEL
LIN {X 0,Y 249.245,Z 614.436,A -85,B 0,C 180,E1 -19006.38,E2 -19006.38} C_VEL
